(* CODESYS project CtaAppModBus_2.0.0.3.library
   Description: Modbus Library der CTA
   Version: 2.0.0.3
   Title: CtaAppModbus
   Author: SIS
   Company: CTA
   Placeholder: CtaAppModbus
   DocFormat: reStructuredText
   CompiledLibraryCompatibilityVersion: CODESYS V3.5 SP16 Patch 3
   LanguageModelAttribute: qualified-access-only
   DefaultNamespace: CtaAppModbus

Project tree, tasks and I/O mapping:
  libraries: Standard, 3.5.18.0 (System); CtaVisSymbols, 2.0.0.1 (CTA); CtaSysConfig, 2.0.0.0 (CTA); CtaAppTime, 2.0.0.0 (CTA); CtaAppBmk, 2.0.0.0 (CTA); VisuSymbols, 4.5.0.0 (System); VisuDialogs, * (System); ModbusFB, 4.5.0.0 (CODESYS); CtaVisUser, 1.0.0.0 (CTA); Util, 3.5.19.0 (System)
  10 Documenation/
    global variables VersionHistory
    global variables readMe
  00000000-0000-0000-0000-000000000000|D:\CoDeSys\LibrariesV3\trunk\Intern\CAA\CAA Template\3.4.0.0 draft\Placeholder.xml
  00000000-0000-0000-0000-000000000000|D:\CoDeSys\LibrariesV3\trunk\Intern\CAA\CAA Template\3.2.0.3 draft\Prefix.pdf
  00000000-0000-0000-0000-000000000000|D:\CoDeSys\LibrariesV3\trunk\Intern\CAA\CAA Template\3.5.2.0 draft\Placeholder.xml
  20 Structs/
    CLIENT/
      NETWORK/
        data type scTcpClientParameter
      SERIAL/
        data type scSerialPortParameter
        data type scSerialClientParameter
    SERVER/
      PARAMETER/
        SERIAL/
          data type scSerial
        data type scModBusServerParameter
        TCP/
          data type scTcp
  21 Interface/
    CLIENTMANAGER/
      BASE/
        interface ITF_MB_CLIENTMANAGER: AY_ITF_MBCLIENT_VIS, ITF_BASE_CLIENT, OperationTime, RELOAD_ARRAY
      RTU/
        interface ITF_MB_CLIENTMANAGER_RTU: P_fbbyDataBits, P_fbdwBaudrate, P_fbenDTRControl, P_fbenParity, P_fbenPort, P_fbenStopBits, P_fbenRTSControl, P_fbxRtuAscii
      TCP/
        interface ITF_MB_CLIENTMANAGER_TCP
    MBJOB/
      interface ITF_MBJOB: DESTROY, PARENT, pByte, SELF, BIG_SYBIL, byMbFunction, LOW_SYBIL, wMbAdress, wQuantity
    CLIENT/
      TCP/
        interface ITF_MB_CLIENT_TCP: WRITE_DELAY, IP_ADRESS, NODE_ID, P_fbstIpAdress, P_fbtReadDelay, P_fbtTimeOut, P_fbtWriteDelay, P_fbuiPort, P_fbusiNodeId, P_fbxEnable, PORT, READ_DELAY, TIMEOUT, ConnectTcp, Connected, ClientTcp
      RTU/
        interface ITF_MB_CLIENT_RTU: TIMEOUT, WRITE_DELAY, NODE_ID, P_fbtReadDelay, P_fbtWriteDelay, P_fbusiNodeId, P_fbxEnable, P_fbtTimeOut, READ_DELAY
      BASE/
        interface ITF_CLIENT: AY_ITF_MBJOB_VIS, COUNT, CREATE_JOB, RELOAD_ARRAY, DESTROY_JOB, SELF, ERROR_ID, ERROR, AllJobsDone, ADD_MODBUS_JOB, CALL_AFTER_LAST_JOB_DONE, CHECK_IF_JOB_EXIST, BASE_MBJOB, ExecuteTime, EXEPTION_CODE, GET_NEXT_JOB, GET_READY, IsCurrentCall, LOW_SYBIL, BIG_SYBIL, CONFIRM_ALL_JOBS_DONE, ENABLE, DESTROY_ALL_JOBS_ACTIVE, DESTROY_ALL_JOBS_REQUEST
    SERVER/
      interface ITF_SERVER_INFO_PARA: P_Serial_fbxRtuAscii, P_Serial_fbbyDataBits, NoSerialAccesSince, P_Serial_fbenDTRControl, P_Serial_fbenParity, P_Serial_fbenStopBits, P_Serial_fbenPort, P_Serial_fbtWatchDog, P_Serial_fbenRTSControl, P_Serial_fbxEnableWatchDog, P_Serial_fbusiNodeId, P_Serial_fbxEnable, P_Serial_fbdwBaudrate, TimeOutSerialWatchDog, RequestDataSerial, NoTcpAccesSince, P_Tcp_fbstInterface, P_Tcp_fbtWatchDog, P_Tcp_fbxEnable, P_Tcp_fbxEnableWatchDog, RequestDataTcp, TimeOutTcpWatchDog, P_Tcp_fbwPort, P_LoggingOp
      interface ITF_SERVER: metSetInputRegister, metSetHoldingRegister, metGetCoil, metGetHoldingRegister, metSetCoil, metSetDiscretInput
  30 Program Organization Units/
    FC/
      function fcStringIPtoByteArray [ST]
      function fcCheckIp [ST]
      function FcBytePointToBoolValue [ST]
      function FcBytePointToWordValue [ST]
      function fcSetInitialIPString [ST]
    CLIENT/
      BASE/
        function block FB_MB_CLIENT [ST]: ENABLE, ADD_MODBUS_JOB, COUNT, CREATE_JOB, DESTROY_JOB, ERROR, BIG_SYBIL, CALL_AFTER_LAST_JOB_DONE, CHECK_IF_JOB_EXIST, CONFIRM_ALL_JOBS_DONE, AllJobsDone, AY_ITF_MBJOB_VIS, BASE_MBJOB, ERROR_ID, ExecuteTime, EXEPTION_CODE, GET_NEXT_JOB, GET_READY, IsCurrentCall, LOW_SYBIL, RELOAD_ARRAY, SELF, DESTROY_ALL_JOBS_REQUEST, DESTROY_ALL_JOBS_ACTIVE, DESTROY_ALL_JOBS
      RTU/
        function block FB_MB_CLIENT_RTU [ST]: actConfig, ENABLE, NODE_ID, P_fbtReadDelay, P_fbtTimeOut, P_fbtWriteDelay, P_fbusiNodeId, P_fbxEnable, READ_DELAY, TIMEOUT, WRITE_DELAY
      TCP/
        function block FB_MB_CLIENT_TCP [ST]: actConfig, ENABLE, IP_ADRESS, P_fbtTimeOut, P_fbtWriteDelay, P_fbuiPort, P_fbusiNodeId, P_fbxEnable, WRITE_DELAY, PORT, NODE_ID, P_fbstIpAdress, READ_DELAY, P_fbtReadDelay, TIMEOUT, ConnectTcp, Connected, ClientTcp
        function block FB_MB_CLIENT_TCP_1 [ST]: actConfig, ENABLE, IP_ADRESS, P_fbtReadDelay, P_fbtTimeOut, P_fbtWriteDelay, P_fbuiPort, P_fbusiNodeId, P_fbxEnable, WRITE_DELAY, PORT, NODE_ID, P_fbstIpAdress, READ_DELAY, TIMEOUT
    SERVER/
      function block FB_SERVER [ST]: actConfig, actDataModel, actSerial, actTcp, metGetCoil, metGetHoldingRegister, metSetCoil, metSetDiscretInput, metSetHoldingRegister, metSetInputRegister, P_Serial_fbxEnableWatchDog, P_Serial_fbxRtuAscii, NoSerialAccesSince, P_Serial_fbbyDataBits, P_Serial_fbdwBaudrate, P_Serial_fbenDTRControl, P_Serial_fbenParity, P_Serial_fbenPort, P_Serial_fbenRTSControl, P_Serial_fbenStopBits, P_Serial_fbtWatchDog, P_Serial_fbusiNodeId, P_Serial_fbxEnable, RequestDataSerial, TimeOutSerialWatchDog, TimeOutTcpWatchDog, P_Tcp_fbwPort, P_Tcp_fbxEnable, P_Tcp_fbxEnableWatchDog, RequestDataTcp, NoTcpAccesSince, P_Tcp_fbstInterface, P_Tcp_fbtWatchDog, P_LoggingOp
      function block fbModBusServer [ST]: actConfig, actModBusServerSerial, actModBusServerTcp, actModBusServerUdp, metAddSerialControll, metAddTcpControll, metAddUdpControll, metGetCoil, metGetHoldingRegister, metSetCoil, metSetDiscretInput, metSetHoldingRegister, metSetInputRegister
      Serial/
        function block ServerSerial_Extended [ST]: RequestData, ProcessMaskWriteRegister, ProcessReadCoils, ProcessReadDiscreteInputs, ProcessReadHoldingRegisters, ProcessReadInputRegisters, ProcessReadWriteMultipleRegisters, ProcessWriteMultipleCoils, ProcessWriteMultipleRegisters, ProcessWriteSingleCoil, ProcessWriteSingleRegister
      Tcp/
        function block ServerTCP_Extended [ST]: RequestData, ProcessMaskWriteRegister, ProcessReadCoils, ProcessReadDiscreteInputs, ProcessReadHoldingRegisters, ProcessReadInputRegisters, ProcessReadWriteMultipleRegisters, ProcessWriteMultipleCoils, ProcessWriteMultipleRegisters, ProcessWriteSingleCoil, ProcessWriteSingleRegister
    MBJOB/
      function block FB_MBJOB [ST]: wMbAdress, BIG_SYBIL, wQuantity, SELF, byMbFunction, DESTROY, LOW_SYBIL, PARENT, pByte
    CLIENTMANAGER/
      RTU/
        function block FB_MB_CLIENTMANAGER_RTU [ST]: actCallFunctions, actDelays, actConfig, actExecuteFunction, actGetError, P_fbbyDataBits, P_fbdwBaudrate, P_fbenDTRControl, P_fbenParity, P_fbenRTSControl, P_fbenStopBits, P_fbxRtuAscii, P_fbenPort, actCheckBusy
      TCP/
        function block FB_MB_CLIENTMANAGER_TCP [ST]: actCallFunctions, actCheckBusy, actDelays, actExecuteFunction, actGetError
        function block FB_MB_CLIENTMANAGER_TCP_1 [ST]: actCallFunctions, actCheckBusy, actDelays, actExecuteFunction, actGetError
      BASE/
        function block FB_MB_CLIENTMANAGER [ST]: RELOAD_ARRAY, ADD_MODBUS_CLIENT, CHECK_IF_EXIST, AY_ITF_MBCLIENT_VIS, ITF_BASE_CLIENT, OperationTime, COUNT_ENABLED
  40 Visualizations/
    CLIENT/
      CLIENT/
        visualisation DIA_CLIENT
        JOBS/
          visualisation VIS_CLIENT_JOBS
          visualisation VIS_CLIENT_JOBS_QUERRY
          visualisation VIS_CLIENT_JOBS_TABLE
        MENÜ/
          visualisation VIS_CLIENT_MENÜ
        OVERWIEV/
          visualisation VIS_CLIENT_OVERWIEV
          visualisation VIS_CLIENT_OVERWIEV_QUERY
        PARAMETER/
          visualisation VIS_CLIENT_PARAMETER
      RTU/
        PARAMETER/
          visualisation VIS_CLIENT_PARAMETER_RTU_QUERY
          visualisation VIS_CLIENT_PARAMETER_RTU
          visualisation VIS_CLIENT_PARAMETER_RTU_TEMP
      TCP/
        PARAMETER/
          visualisation VIS_CLIENT_PARAMETER_TCP
          visualisation VIS_CLIENT_PARAMETER_TCP_TEMP
          visualisation VIS_CLIENT_PARAMETER_TCP_QUERY
    TEXTLIST/
      text list TEXT_DTR_CONTROL
      text list TEXT_PARITY
      text list TEXT_RTS_CONTROL
      text list TEXT_STOPBITS
      text list TXT_COMPORT
    CLIENTMANAGER/
      visualisation DIA_CLIENT_MANAGER
      LINE/
        visualisation VIS_CLIENT_LINE
        visualisation VIS_CLIENT_LINE_QUERRY
      MENÜ/
        visualisation VIS_CLIENTMANAGER_MENÜ
      OVERWIEV/
        visualisation VIS_CLIENT_MANAGER_OVERWIEV
        visualisation VIS_CLIENT_MANAGER_OVERWIEV_QUERRY
        visualisation VIS_CLIENT_MANAGER_TABLE
      PARAMETER/
        visualisation VIS_CLIENT_MANAGER_PARAMETER
      RTU/
        PARAMETER/
          visualisation VIS_CLIENT_MANAGER_PARAMETER_RTU
          visualisation VIS_CLIENT_MANAGER_PARAMETER_RTU_QUERY
          visualisation VIS_CLIENT_MANAGER_PARAMETER_RTU_TEMP
      TCP/
        PARAMETER/
          visualisation VIS_CLIENT_MANAGER_PARAMETER_TCP
          visualisation VIS_CLIENT_MANAGER_PARAMETER_TCP_QUERY
    HELPER/
      visualisation VIS_IP_PARAMETER
      visualisation DIA_IP_INPUT
      visualisation VIS_IP_PARAMETER_QUERRY
      visualisation VIS_IP_PARAMETER_BASE
    MBJOB/
      visualisation VIS_JOB
      visualisation VIS_JOB_QUERRY
    SERVER/
      visualisation DIA_SERVER
      SERIAL/
        visualisation VIS_SERVER_SERIAL_STATE
        visualisation VIS_SERVER_SERIAL_STATE_INFO
        PARAMETER/
          visualisation DIA_SERVER_SERIAL_PARAMETER
          visualisation VIS_SERVER_SERIAL_PARAMETER
      TCP/
        visualisation VIS_SERVER_TCP_STATE
        visualisation VIS_SERVER_TCP_STATE_INFO
        PARAMETER/
          visualisation DIA_SERVER_TCP_PARAMETER
          visualisation VIS_SERVER_TCP_PARAMETER
  text list GlobalTextList
  60 Textlisten/
    SERIAL/
      text list txtHandshake
      text list txtParity
      text list txtPhysikalLayer
      text list txtStopBits
    text list txtLoggingOp
*)

// 20 Structs/CLIENT/SERIAL/scSerialPortParameter
TYPE scSerialPortParameter :
    STRUCT 
		fbenPort							:	CtaSysConfig.fbINT;			// PORT NONE , COM1, COM2 ...
		fbdwBaudrate						:	CtaSysConfig.fbDWORD;		// Baudrate 
		fbbyDataBits						:	CtaSysConfig.fbBYTE;		// Data Bits
		fbenParity							:	CtaSysConfig.fbBYTE;		// Parity
		fbenStopBits						:	CtaSysConfig.fbBYTE;		// Stopbits
		fbenDTRControl						:	CtaSysConfig.fbBYTE;		// DTR Control
		fbenRTSControl						:	CtaSysConfig.fbBYTE;		// RTS Control
		fbxRtuAscii							:	CtaSysConfig.fbBOOL;		// RTU = FALSE , ASCII = TRUE
    END_STRUCT
END_TYPE

// 20 Structs/CLIENT/SERIAL/scSerialClientParameter
TYPE scSerialClientParameter :
    STRUCT
        fbxEnable					:	CtaSysConfig.fbBOOL;       // Serial Server Enable        
        fbusiNodeId					:	CtaSysConfig.fbUSINT;      // Serial Server Id        
        fbtTimeOut					:	CtaSysConfig.fbTIME;       // Timeout Time
		fbtReadDelay				:	CtaSysConfig.fbTIME; 	   // Read Delay
		fbtWriteDelay				:	CtaSysConfig.fbTIME;	   // Write Delay
    END_STRUCT
END_TYPE

// 20 Structs/SERVER/PARAMETER/SERIAL/scSerial
TYPE scSerial :
    STRUCT
        fbxEnable           				:   CtaSysConfig.fbBOOL;        // Serial Server Enable
        fbxEnableWatchDog   				:   CtaSysConfig.fbBOOL;        // WatchDog Enable
        fbtWatchDog         				:   CtaSysConfig.fbTIME;        // WatchDog Time		
		fbenPort							:	CtaSysConfig.fbINT;			// PORT NONE , COM1, COM2 ...
		fbusiNodeId							:	CtaSysConfig.fbUSINT;      	// Serial Server Id  
		fbdwBaudrate						:	CtaSysConfig.fbDWORD;		// Baudrate 
		fbbyDataBits						:	CtaSysConfig.fbBYTE;		// Data Bits
		fbenParity							:	CtaSysConfig.fbBYTE;		// Parity
		fbenStopBits						:	CtaSysConfig.fbBYTE;		// Stopbits
		fbenDTRControl						:	CtaSysConfig.fbBYTE;		// DTR Control
		fbenRTSControl						:	CtaSysConfig.fbBYTE;		// RTS Control
		fbxRtuAscii							:	CtaSysConfig.fbBOOL;		// RTU = FALSE , ASCII = TRUE
    END_STRUCT
END_TYPE

// 20 Structs/SERVER/PARAMETER/TCP/scTcp
TYPE scTcp :
    STRUCT
        fbxEnable           :   CtaSysConfig.fbBOOL;           // Tcp Server Enable    
        fbwPort             :   CtaSysConfig.fbWORD;           // Tcp Server Port
        fbxEnableWatchDog   :   CtaSysConfig.fbBOOL;           // WatchDog Enable
        fbtWatchDog         :   CtaSysConfig.fbTIME;           // WatchDog Time
		fbstInterface		:	CtaSysConfig.fbSTRING40;	   // Interface Name
    END_STRUCT
END_TYPE

// 20 Structs/CLIENT/NETWORK/scTcpClientParameter
TYPE scTcpClientParameter :
    STRUCT
        fbxEnable					:	CtaSysConfig.fbBOOL;        // Serial Server Enable       
        fbusiNodeId					:	CtaSysConfig.fbUSINT;     	// Serial Server Id  
        fbtTimeOut					:	CtaSysConfig.fbTIME;        // Timeout Time
        fbtReadDelay				:	CtaSysConfig.fbTIME;      	// Read Delay        
        fbtWriteDelay				:	CtaSysConfig.fbTIME;     	// Write Delay 	
		fbuiPort					:	CtaSysConfig.fbUINT;      	// Port Nr  
		fbstIpAdress				:	CtaSysConfig.fbSTRING40;    // IP Adresse   
    END_STRUCT
END_TYPE

// 20 Structs/SERVER/PARAMETER/scModBusServerParameter
TYPE scModBusServerParameter :
    STRUCT
        scSerial    :   scSerial;
        scTcp       :   scTcp;
		loggingOp	:	CtaSysConfig.fbDWORD;
    END_STRUCT
END_TYPE

// 10 Documenation/VersionHistory
(* 

.. image:: ../../Images/CTA_Logo.jpg
   :align: right
   :width: 15% 

**Vorlage**   


============ =========== =========== ============================================
**Date**     **Version** **Author**  **Change**
------------ ----------- ----------- --------------------------------------------
04.03.2021   0.0.0.0     SIS         Vorlage erstellt

============ =========== =========== ============================================


*)
VAR_GLOBAL
    stInfo : STRING:= '0.0.0.0, Vorlage, CTA';
END_VAR

// 10 Documenation/readMe
(*

**ReadMe**
 
|	**Empfehlung**
|
|	Dokumentrieren Sie die Library für eine nachhaltige Entwicklung
|     
| *Beispiel* 
|
| Dies ist die Vorlage Library der CTA. Erstellen Sie ihre Library anhand dieser Vorlage.
*)

VAR_GLOBAL
    xReadMeDone              :   BOOL;
END_VAR

// 21 Interface/SERVER/ITF_SERVER_INFO_PARA
INTERFACE ITF_SERVER_INFO_PARA EXTENDS ITF_SERVER

PROPERTY P_Serial_fbxRtuAscii : CtaSysConfig.ITF_BOOL
GET
END_GET
END_PROPERTY

PROPERTY P_Serial_fbbyDataBits : CtaSysConfig.ITF_BYTE
GET
END_GET
END_PROPERTY

PROPERTY NoSerialAccesSince : TIME
GET
END_GET
END_PROPERTY

PROPERTY P_Serial_fbenDTRControl : CtaSysConfig.ITF_BYTE
GET
END_GET
END_PROPERTY

PROPERTY P_Serial_fbenParity : CtaSysConfig.ITF_BYTE
GET
END_GET
END_PROPERTY

PROPERTY P_Serial_fbenStopBits : CtaSysConfig.ITF_BYTE
GET
END_GET
END_PROPERTY

PROPERTY P_Serial_fbenPort : CtaSysConfig.ITF_INT
GET
END_GET
END_PROPERTY

PROPERTY P_Serial_fbtWatchDog : CtaSysConfig.ITF_TIME
GET
END_GET
END_PROPERTY

PROPERTY P_Serial_fbenRTSControl : CtaSysConfig.ITF_BYTE
GET
END_GET
END_PROPERTY

PROPERTY P_Serial_fbxEnableWatchDog : CtaSysConfig.ITF_BOOL
GET
END_GET
END_PROPERTY

PROPERTY P_Serial_fbusiNodeId : CtaSysConfig.ITF_USINT
GET
END_GET
END_PROPERTY

PROPERTY P_Serial_fbxEnable : CtaSysConfig.ITF_BOOL
GET
END_GET
END_PROPERTY

PROPERTY P_Serial_fbdwBaudrate : CtaSysConfig.ITF_DWORD
GET
END_GET
END_PROPERTY

PROPERTY TimeOutSerialWatchDog : BOOL
GET
END_GET
END_PROPERTY

PROPERTY RequestDataSerial : String
GET
END_GET
END_PROPERTY

PROPERTY NoTcpAccesSince : TIME
GET
END_GET
END_PROPERTY

PROPERTY P_Tcp_fbstInterface : CtaSysConfig.ITF_STRING40
GET
END_GET
END_PROPERTY

PROPERTY P_Tcp_fbtWatchDog : CtaSysConfig.ITF_TIME
GET
END_GET
END_PROPERTY

PROPERTY P_Tcp_fbxEnable : CtaSysConfig.ITF_BOOL
GET
END_GET
END_PROPERTY

PROPERTY P_Tcp_fbxEnableWatchDog : CtaSysConfig.ITF_BOOL
GET
END_GET
END_PROPERTY

PROPERTY RequestDataTcp : STRING
GET
END_GET
END_PROPERTY

PROPERTY TimeOutTcpWatchDog : BOOL
GET
END_GET
END_PROPERTY

PROPERTY P_Tcp_fbwPort : CtaSysConfig.ITF_WORD
GET
END_GET
END_PROPERTY

PROPERTY P_LoggingOp : CtaSysConfig.ITF_DWORD
GET
END_GET
END_PROPERTY

END_INTERFACE

// 21 Interface/SERVER/ITF_SERVER
INTERFACE ITF_SERVER EXTENDS __SYSTEM.IQueryInterface

METHOD metSetInputRegister : BOOL
VAR_INPUT
    wAdr          : WORD;
    wValue        : WORD;
END_VAR
END_METHOD

METHOD metSetHoldingRegister : BOOL
VAR_INPUT
    wAdr          : WORD;
    wValue        : WORD;
END_VAR
END_METHOD

METHOD metGetCoil : BOOL
VAR_INPUT
    wAdr          : WORD;
END_VAR
END_METHOD

METHOD metGetHoldingRegister : WORD
VAR_INPUT
    wAdr          : WORD;
END_VAR
END_METHOD

METHOD metSetCoil : BOOL
VAR_INPUT
    wAdr          : WORD;
    xValue        : BOOL;
END_VAR
END_METHOD

METHOD metSetDiscretInput : BOOL
VAR_INPUT
    wAdr          : WORD;
    xValue        : BOOL;
END_VAR
END_METHOD

END_INTERFACE

// 21 Interface/CLIENTMANAGER/BASE/ITF_MB_CLIENTMANAGER
INTERFACE ITF_MB_CLIENTMANAGER EXTENDS CtaAppBmk.ITF_BMK

PROPERTY AY_ITF_MBCLIENT_VIS : ARRAY[0..9] OF ITF_CLIENT
GET
END_GET
END_PROPERTY

PROPERTY ITF_BASE_CLIENT : ITF_CLIENT
GET
END_GET
END_PROPERTY

PROPERTY OperationTime : LTIME
GET
END_GET
END_PROPERTY

METHOD RELOAD_ARRAY
VAR_INPUT
	xInit				:	BOOL;
	xLoadNext10			:	BOOL;
	xLoadLast10			:	BOOL;
END_VAR
END_METHOD

END_INTERFACE

// 21 Interface/CLIENT/BASE/ITF_CLIENT
INTERFACE ITF_CLIENT  EXTENDS CtaAppBmk.ITF_BMK

PROPERTY AY_ITF_MBJOB_VIS : ARRAY[0..9] OF ITF_MBJOB
GET
END_GET
END_PROPERTY

PROPERTY COUNT : UINT
GET
END_GET
END_PROPERTY

METHOD CREATE_JOB : BOOL
VAR_INPUT
	_byMbFunction	:	BYTE;
	_wMbAdress		:	WORD;
	_pData			:	POINTER TO BYTE;
	_wQuantity		:	WORD;		
END_VAR
END_METHOD

METHOD RELOAD_ARRAY
VAR_INPUT
	xInit				:	BOOL;
	xLoadNext10			:	BOOL;
	xLoadLast10			:	BOOL;
END_VAR
END_METHOD

METHOD DESTROY_JOB : BOOL
VAR_INPUT
	_byMbFunction	:	BYTE;
	_wMbAdress		:	WORD;
	_pData			:	POINTER TO BYTE;
	_wQuantity		:	WORD;		
END_VAR
END_METHOD

PROPERTY SELF : ITF_CLIENT
GET
END_GET
END_PROPERTY

PROPERTY ERROR_ID : ModbusFB.Error
GET
END_GET
SET
END_SET
END_PROPERTY

PROPERTY ERROR : BOOL
GET
END_GET
SET
END_SET
END_PROPERTY

PROPERTY AllJobsDone : BOOL
GET
END_GET
END_PROPERTY

METHOD ADD_MODBUS_JOB
VAR_INPUT
	ITF_MBJOB_IN	:	ITF_MBJOB;
END_VAR
END_METHOD

METHOD CALL_AFTER_LAST_JOB_DONE
VAR_INPUT
END_VAR
END_METHOD

METHOD CHECK_IF_JOB_EXIST : BOOL
VAR_INPUT
	_byMbFunction	:	BYTE;
	_wMbAdress		:	WORD;
	_pByte			:	POINTER TO BYTE;
	_wQuantity		:	WORD;	
END_VAR
END_METHOD

PROPERTY BASE_MBJOB : ITF_MBJOB
GET
END_GET
END_PROPERTY

PROPERTY ExecuteTime : LTIME
GET
END_GET
END_PROPERTY

PROPERTY EXEPTION_CODE : ModbusFB.ExceptionCodes
GET
END_GET
SET
END_SET
END_PROPERTY

METHOD GET_NEXT_JOB : BOOL
VAR_OUTPUT
	_byMbFunction	:	BYTE;
	_wMbAdress		:	WORD;
	_pByte			:	POINTER TO BYTE;
	_wQuantity		:	WORD;	
END_VAR
END_METHOD

METHOD GET_READY : BOOL
VAR_INPUT
END_VAR
END_METHOD

PROPERTY IsCurrentCall : BOOL
GET
END_GET
END_PROPERTY

PROPERTY LOW_SYBIL : ITF_CLIENT
SET
END_SET
GET
END_GET
END_PROPERTY

PROPERTY BIG_SYBIL : ITF_CLIENT
GET
END_GET
SET
END_SET
END_PROPERTY

PROPERTY CONFIRM_ALL_JOBS_DONE : BOOL
GET
END_GET
END_PROPERTY

PROPERTY ENABLE : BOOL
GET
END_GET
END_PROPERTY

PROPERTY DESTROY_ALL_JOBS_ACTIVE : BOOL
GET
END_GET
END_PROPERTY

METHOD DESTROY_ALL_JOBS_REQUEST
VAR_INPUT
END_VAR
END_METHOD

END_INTERFACE

// 21 Interface/MBJOB/ITF_MBJOB
INTERFACE ITF_MBJOB EXTENDS __System.IQUERYINTERFACE

METHOD DESTROY
END_METHOD

PROPERTY PARENT : ITF_CLIENT
SET
END_SET
END_PROPERTY

PROPERTY pByte : POINTER TO BYTE
GET
END_GET
SET
END_SET
END_PROPERTY

PROPERTY SELF : ITF_MBJOB
GET
END_GET
END_PROPERTY

PROPERTY BIG_SYBIL : ITF_MBJOB
GET
END_GET
SET
END_SET
END_PROPERTY

PROPERTY byMbFunction : BYTE
GET
END_GET
SET
END_SET
END_PROPERTY

PROPERTY LOW_SYBIL : ITF_MBJOB
GET
END_GET
SET
END_SET
END_PROPERTY

PROPERTY wMbAdress : WORD
GET
END_GET
SET
END_SET
END_PROPERTY

PROPERTY wQuantity : WORD
GET
END_GET
SET
END_SET
END_PROPERTY

END_INTERFACE

// 21 Interface/CLIENTMANAGER/RTU/ITF_MB_CLIENTMANAGER_RTU
INTERFACE ITF_MB_CLIENTMANAGER_RTU EXTENDS ITF_MB_CLIENTMANAGER

PROPERTY P_fbbyDataBits : CtaSysConfig.ITF_DATATYPE
GET
END_GET
END_PROPERTY

PROPERTY P_fbdwBaudrate : CtaSysConfig.ITF_DATATYPE
GET
END_GET
END_PROPERTY

PROPERTY P_fbenDTRControl : CtaSysConfig.ITF_BYTE
GET
END_GET
END_PROPERTY

PROPERTY P_fbenParity : CtaSysConfig.ITF_BYTE
GET
END_GET
END_PROPERTY

PROPERTY P_fbenPort : CtaSysConfig.ITF_INT
GET
END_GET
END_PROPERTY

PROPERTY P_fbenStopBits : CtaSysConfig.ITF_BYTE
GET
END_GET
END_PROPERTY

PROPERTY P_fbenRTSControl : CtaSysConfig.ITF_BYTE
GET
END_GET
END_PROPERTY

PROPERTY P_fbxRtuAscii : CtaSysConfig.ITF_DATATYPE
GET
END_GET
END_PROPERTY

END_INTERFACE

// 21 Interface/CLIENT/TCP/ITF_MB_CLIENT_TCP
INTERFACE ITF_MB_CLIENT_TCP  EXTENDS ITF_CLIENT

PROPERTY WRITE_DELAY : TIME
GET
END_GET
END_PROPERTY

PROPERTY IP_ADRESS : STRING(15)
GET
END_GET
END_PROPERTY

PROPERTY NODE_ID : USINT
GET
END_GET
END_PROPERTY

PROPERTY P_fbstIpAdress : CtaSysConfig.ITF_DATATYPE
GET
END_GET
END_PROPERTY

PROPERTY P_fbtReadDelay : CtaSysConfig.ITF_DATATYPE
GET
END_GET
END_PROPERTY

PROPERTY P_fbtTimeOut : CtaSysConfig.ITF_DATATYPE
GET
END_GET
END_PROPERTY

PROPERTY P_fbtWriteDelay : CtaSysConfig.ITF_DATATYPE
GET
END_GET
END_PROPERTY

PROPERTY P_fbuiPort : CtaSysConfig.ITF_DATATYPE
GET
END_GET
END_PROPERTY

PROPERTY P_fbusiNodeId : CtaSysConfig.ITF_DATATYPE
GET
END_GET
END_PROPERTY

PROPERTY P_fbxEnable : CtaSysConfig.ITF_DATATYPE
GET
END_GET
END_PROPERTY

PROPERTY PORT : UINT
GET
END_GET
END_PROPERTY

PROPERTY READ_DELAY : TIME
GET
END_GET
END_PROPERTY

PROPERTY TIMEOUT : TIME
GET
END_GET
END_PROPERTY

METHOD ConnectTcp : BOOL
VAR_INPUT
END_VAR
END_METHOD

PROPERTY Connected : BOOL
GET
END_GET
END_PROPERTY

PROPERTY  ClientTcp : REFERENCE TO ModbusFB.Client
GET
END_GET
END_PROPERTY

END_INTERFACE

// 30 Program Organization Units/FC/fcStringIPtoByteArray
FUNCTION fcStringIPtoByteArray : ARRAY[0..3] OF BYTE
VAR_INPUT
	stIP	:	STRING;
END_VAR
VAR
    temp_string 	: STRING;
    dot_pos 		: INT;
    i 				: INT;
    part 			: STRING[4];
    value 			: WORD;
END_VAR

temp_string := stIP;
REPEAT
    dot_pos := FIND(temp_string,'.');
    IF dot_pos > 0 THEN
        part := LEFT(temp_string, dot_pos - 1);
        temp_string := RIGHT(temp_string, LEN(temp_string) - dot_pos);
    ELSE
        part := temp_string;
    END_IF

    // Umwandeln in BYTE
    value := STRING_TO_WORD(part);
    IF (value >= 0) AND (value <= 255) THEN
        fcStringIPtoByteArray[i] := WORD_TO_BYTE(value);
    ELSE
        RETURN;
    END_IF

    i := i + 1;
UNTIL (dot_pos = 0) OR (i > 3)
END_REPEAT

// Setze auf 0 wenn nicht 4 Segmente gefunden wurden
IF i <> 4 THEN
	fcStringIPtoByteArray[0] := 0;
	fcStringIPtoByteArray[1] := 0;
	fcStringIPtoByteArray[2] := 0;
	fcStringIPtoByteArray[3] := 0;
END_IF

END_FUNCTION

// 30 Program Organization Units/FC/fcCheckIp
FUNCTION fcCheckIp : BOOL
VAR_INPUT
    stIp           : STRING[20];
END_VAR
VAR
    iFor           : INT;
    iCountPacket   : INT;
    iCountPoint    : INT;
    iCountZiffer   : INT;
    xFail          : BOOL;
END_VAR

FOR iFor := LEN(stIp) TO 0 BY -1 DO
    // Check Termination
    IF iFor = LEN(stIp) THEN
        IF stIp[iFor] <> 0 THEN 
            xFail := TRUE; // No Termination
            EXIT;       
        END_IF;
	ELSE
        // Check if Ziffer
        IF stIp[iFor] >= 48 AND stIp[iFor] <= 57 THEN    
            IF iCountZiffer < 3 THEN
                IF iCountZiffer = 0 THEN
                    IF iFor >= 2 THEN
                        IF stIp[iFor - 2] >= 50 THEN
                            // Check if Ziffer <= 5
                            IF stIp[iFor] <= 53 THEN     
                                iCountZiffer := iCountZiffer + 1;
                            ELSE
                                xFail := TRUE;  // Max is 255
                                EXIT;
                            END_IF;   
                        ELSE
                            iCountZiffer := iCountZiffer + 1;                   
						END_IF;                        
                    ELSE
                        iCountZiffer := iCountZiffer + 1;
					END_IF
                ELSIF iCountZiffer = 1 THEN
                    IF iFor <> 0 THEN
                        IF stIp[iFor - 1] = 46 THEN
                            iCountZiffer := iCountZiffer + 1;
                        // Check if next Ziffer is 2    
                        ELSIF stIp[iFor - 1] >= 50 THEN  
                            // Check if Ziffer <= 5
                            IF stIp[iFor] <= 53 THEN     
                                iCountZiffer := iCountZiffer + 1;
                            ELSE
                                xFail := TRUE;  // Max is 255
                                EXIT;
                            END_IF;    
                        END_IF;
                    ELSE
                        iCountZiffer := iCountZiffer + 1;        
					END_IF;                       
                ELSIF iCountZiffer = 2 THEN
                    IF stIp[iFor] <= 50 THEN
                        iCountZiffer := iCountZiffer + 1;
                    ELSE
                        xFail := TRUE;
                        EXIT;
					END_IF
                END_IF;    
            ELSIF iCountZiffer = 3 THEN
                xFail := TRUE; // More Then 3 Ziffers not allowed!
                EXIT;
            END_IF;
        // Check if Point
        ELSIF stIp[iFor] = 46 THEN
            IF iCountZiffer > 0 THEN
                iCountPacket := iCountPacket + 1;
                iCountPoint  := iCountPoint + 1;
                iCountZiffer := 0;
            ELSE
                xFail := TRUE; // Empty Packet not allowed!
                EXIT;
            END_IF;   
        END_IF;
    END_IF;
END_FOR;

IF xFail THEN
    fcCheckIp := FALSE;
ELSIF iCountPoint = 3 AND iCountPacket = 3 AND iCountZiffer > 0 THEN    
    fcCheckIp := TRUE;
END_IF;

END_FUNCTION

// 30 Program Organization Units/CLIENTMANAGER/TCP/FB_MB_CLIENTMANAGER_TCP
{attribute 'no_assign'}
FUNCTION_BLOCK FB_MB_CLIENTMANAGER_TCP EXTENDS FB_MB_CLIENTMANAGER IMPLEMENTS ITF_MB_CLIENTMANAGER_TCP
VAR_OUTPUT
END_VAR
VAR
	_TEMP_MBU_CLIENT_TCP				:	ITF_MB_CLIENT_TCP;
	
	fbReadCoilsFc01						:	ModbusFB.ClientRequestReadCoils;
	fbReadDiscreteInputsFc02			:	ModbusFB.ClientRequestReadDiscreteInputs;
	fbReadHoldingRegistersFc03			:	ModbusFB.ClientRequestReadHoldingRegisters;
	fbReadInputRegistersFc04			:	ModbusFB.ClientRequestReadInputRegisters;
	fbWriteSingleCoilFc05				:	ModbusFB.ClientRequestWriteSingleCoil;
	fbWriteSingleRegisterFc06			:	ModbusFB.ClientRequestWriteSingleRegister;
	fbWriteMultipleCoilsFc15			:	ModbusFB.ClientRequestWriteMultipleCoils;
	fbWriteMultipleRegistersFc16		:	ModbusFB.ClientRequestWriteMultipleRegisters;
	
END_VAR

SUPER^();
(* Check if one is allready Working *)
IF NOT xIsWorking THEN
	(* Get Client Ready *)
	IF __QUERYINTERFACE(_TEMP_MBU_CLIENT,_TEMP_MBU_CLIENT) THEN
		xIsWorking 		:= TRUE;	
		xErrorHappen	:= FALSE;
		eErrorID		:= ModbusFB.Error.OK;
		eExeptionCode	:= ModbusFB.ExceptionCodes.RESPONSE_SUCCESS;		
	(* Get Base Client Ready *)
	ELSIF __QUERYINTERFACE(_BASE_MBU_CLIENT,_TEMP_MBU_CLIENT) THEN
		xIsWorking 		:= TRUE;
		xErrorHappen	:= FALSE;
		eErrorID		:= ModbusFB.Error.OK;
		eExeptionCode	:= ModbusFB.ExceptionCodes.RESPONSE_SUCCESS;
		ltTime 			:= fbTimeStop.Stop();
		fbTimeStop.Start();
	END_IF;
END_IF;
(* Check if is running *)
IF xIsWorking THEN
	IF __QUERYINTERFACE(_TEMP_MBU_CLIENT,_TEMP_MBU_CLIENT) THEN	
		(* Wait until no Execute *)		
		IF 	NOT	fbReadCoilsFc01.xExecute				AND
			NOT	fbReadDiscreteInputsFc02.xExecute	    AND
			NOT	fbReadHoldingRegistersFc03.xExecute     AND
			NOT	fbReadInputRegistersFc04.xExecute	    AND
			NOT	fbWriteSingleCoilFc05.xExecute		    AND
			NOT	fbWriteSingleRegisterFc06.xExecute	    AND
			NOT	fbWriteMultipleCoilsFc15.xExecute	    AND
			NOT	fbWriteMultipleRegistersFc16.xExecute	THEN
			(* Get Type of Port *) 
			IF __QUERYINTERFACE(_TEMP_MBU_CLIENT,_TEMP_MBU_CLIENT_TCP) THEN
				(* Check if Enabled *)
				IF _TEMP_MBU_CLIENT_TCP.ENABLE AND _TEMP_MBU_CLIENT_TCP.COUNT > 0 THEN
					IF NOT _TEMP_MBU_CLIENT_TCP.IsCurrentCall THEN
						_TEMP_MBU_CLIENT_TCP.GET_READY();
						tTimeOut		:= _TEMP_MBU_CLIENT_TCP.TIMEOUT;
						tReadDelay		:= _TEMP_MBU_CLIENT_TCP.READ_DELAY;
						tWriteDelay	 	:= _TEMP_MBU_CLIENT_TCP.WRITE_DELAY;
					END_IF;
					(* Connect *)
					IF NOT _TEMP_MBU_CLIENT_TCP.Connected THEN
						xAbort 			:= _TEMP_MBU_CLIENT_TCP.ConnectTcp();
						usiNodeId 		:= _TEMP_MBU_CLIENT_TCP.NODE_ID;
					END_IF;
				ELSE
					xAbort		:= TRUE;
				END_IF;
			ELSE
				xAbort := TRUE;
			END_IF;
			(* Check if Connected *)
			IF _TEMP_MBU_CLIENT_TCP.Connected AND NOT xAbort THEN
				(* Get Job *)
				IF NOT xTrig THEN
					xTrig := _TEMP_MBU_CLIENT.GET_NEXT_JOB(_byMbFunction => _byMbFunction,_wMbAdress => _wMbAdress,_pByte => _pByte,_wQuantity => _wQuantity);
				END_IF;
				
				(* Delay Function *)
				actDelays();
				
				(* Execute Function *)
				actExecuteFunction();
				
				(* Resett Timer *)
				IF tonDelay.Q THEN
					tonDelay(IN := FALSE);
					xTrig := FALSE;
				END_IF;
			END_IF;
		ELSE
			(* Check Busy *)
			actCheckBusy();					
		END_IF;
		(* Get Errors *)
		actGetError();
		(* Check if All Job as Done *)
		IF _TEMP_MBU_CLIENT.AllJobsDone OR xAbort THEN
			(* Wait until no Execute *)		
			IF 	NOT xTrig									AND
				NOT	fbReadCoilsFc01.xExecute				AND
				NOT	fbReadDiscreteInputsFc02.xExecute	    AND
				NOT	fbReadHoldingRegistersFc03.xExecute     AND
				NOT	fbReadInputRegistersFc04.xExecute	    AND
				NOT	fbWriteSingleCoilFc05.xExecute		    AND
				NOT	fbWriteSingleRegisterFc06.xExecute	    AND
				NOT	fbWriteMultipleCoilsFc15.xExecute	    AND
				NOT	fbWriteMultipleRegistersFc16.xExecute	THEN
				_TEMP_MBU_CLIENT.CALL_AFTER_LAST_JOB_DONE();
				(* Set Error if Job > 0 *)
				IF _TEMP_MBU_CLIENT.COUNT > 0 THEN
					_TEMP_MBU_CLIENT.ERROR			:= xErrorHappen;
					_TEMP_MBU_CLIENT.ERROR_ID		:= eErrorID;
					_TEMP_MBU_CLIENT.EXEPTION_CODE	:= eExeptionCode;
				END_IF;
				_TEMP_MBU_CLIENT 					:= _TEMP_MBU_CLIENT.LOW_SYBIL;
				_byMbFunction 					:= 0;
				_wMbAdress	  					:= 0;
				_pByte		  					:= 0;
				_wQuantity						:= 0;
				xIsWorking						:= FALSE;
				xAbort							:= FALSE;
			END_IF;
		END_IF;
	END_IF;
END_IF;

(* Call Functions *)
actCallFunctions();

ACTION actCallFunctions:
(* Call *)
IF __QUERYINTERFACE(_TEMP_MBU_CLIENT_TCP,_TEMP_MBU_CLIENT_TCP) THEN
	fbReadCoilsFc01(				rClient := _TEMP_MBU_CLIENT_TCP.ClientTcp);		
	fbReadDiscreteInputsFc02(		rClient := _TEMP_MBU_CLIENT_TCP.ClientTcp);  
	fbReadHoldingRegistersFc03(		rClient := _TEMP_MBU_CLIENT_TCP.ClientTcp);
	fbReadInputRegistersFc04(		rClient := _TEMP_MBU_CLIENT_TCP.ClientTcp);	  
	fbWriteSingleCoilFc05(			rClient := _TEMP_MBU_CLIENT_TCP.ClientTcp);	  
	fbWriteSingleRegisterFc06(		rClient := _TEMP_MBU_CLIENT_TCP.ClientTcp);  
	fbWriteMultipleCoilsFc15(		rClient := _TEMP_MBU_CLIENT_TCP.ClientTcp);  
	fbWriteMultipleRegistersFc16(	rClient := _TEMP_MBU_CLIENT_TCP.ClientTcp);
END_IF;
END_ACTION

ACTION actCheckBusy:
(* Reset after Busy *)
fbReadCoilsFc01.xExecute				:= fbReadCoilsFc01.xBusy				;
fbReadDiscreteInputsFc02.xExecute	    := fbReadDiscreteInputsFc02.xBusy		;
fbReadHoldingRegistersFc03.xExecute     := fbReadHoldingRegistersFc03.xBusy		;
fbReadInputRegistersFc04.xExecute	    := fbReadInputRegistersFc04.xBusy		;
fbWriteSingleCoilFc05.xExecute		    := fbWriteSingleCoilFc05.xBusy			;
fbWriteSingleRegisterFc06.xExecute	    := fbWriteSingleRegisterFc06.xBusy		;
fbWriteMultipleCoilsFc15.xExecute	    := fbWriteMultipleCoilsFc15.xBusy		;
fbWriteMultipleRegistersFc16.xExecute   := fbWriteMultipleRegistersFc16.xBusy	;
END_ACTION

ACTION actDelays:
(* Delay Read *)
IF _byMbFunction <= 04 THEN
	tonDelay(IN := xTrig,PT := tReadDelay);
(* Delay Write Single *)
ELSIF _byMbFunction >= 5 AND _byMbFunction <= 6 THEN
	tonDelay(IN := xTrig,PT := tWriteDelay); 
(* Delay Write Multiple *)
ELSIF _byMbFunction >= 15 AND _byMbFunction <= 16 THEN
	tonDelay(IN := xTrig,PT := tWriteDelay); 
ELSE 
	tonDelay(IN := xTrig,PT := T#0MS);
END_IF;
END_ACTION

ACTION actExecuteFunction:
(* Read Coils *)
IF _byMbFunction = 01 THEN
	fbReadCoilsFc01.udiReplyTimeout					:= TO_UDINT(tTimeOut) * 1000; 
	fbReadCoilsFc01.udiTimeOut						:= TO_UDINT(tTimeOut) * 1000 * 2;
	fbReadCoilsFc01.uiUnitId						:= usiNodeId;
	fbReadCoilsFc01.uiStartItem 					:= TO_UINT(_wMbAdress);
	fbReadCoilsFc01.pData 							:= _pByte;
	fbReadCoilsFc01.uiQuantity						:= TO_UINT(_wQuantity);
	fbReadCoilsFc01.xExecute						:= tonDelay.Q;
(* Read Discret Inputs *)                       	
ELSIF _byMbFunction = 02 THEN                   	
	fbReadDiscreteInputsFc02.udiReplyTimeout		:= TO_UDINT(tTimeOut) * 1000; 
	fbReadDiscreteInputsFc02.udiTimeOut				:= TO_UDINT(tTimeOut) * 1000 * 2;
	fbReadDiscreteInputsFc02.uiUnitId				:= usiNodeId;
	fbReadDiscreteInputsFc02.uiStartItem			:= TO_UINT(_wMbAdress);
	fbReadDiscreteInputsFc02.pData 					:= _pByte;
	fbReadDiscreteInputsFc02.uiQuantity				:= TO_UINT(_wQuantity);
	fbReadDiscreteInputsFc02.xExecute				:= tonDelay.Q;
(* Read Holding Registers *)                		
ELSIF _byMbFunction = 03 THEN                   	
	fbReadHoldingRegistersFc03.udiReplyTimeout		:= TO_UDINT(tTimeOut) * 1000; 
	fbReadHoldingRegistersFc03.udiTimeOut			:= TO_UDINT(tTimeOut) * 1000 * 2;
	fbReadHoldingRegistersFc03.uiUnitId				:= usiNodeId;          	
	fbReadHoldingRegistersFc03.uiStartItem			:= TO_UINT(_wMbAdress);
	fbReadHoldingRegistersFc03.pData 				:= _pByte;
	fbReadHoldingRegistersFc03.uiQuantity			:= TO_UINT(_wQuantity);
	fbReadHoldingRegistersFc03.xExecute				:= tonDelay.Q;			
(* Read Input Registers *)	                		
ELSIF _byMbFunction = 04 THEN                   	
	fbReadInputRegistersFc04.udiReplyTimeout		:= TO_UDINT(tTimeOut) * 1000; 
	fbReadInputRegistersFc04.udiTimeOut				:= TO_UDINT(tTimeOut) * 1000 * 2;
	fbReadInputRegistersFc04.uiUnitId				:= usiNodeId;               	
	fbReadInputRegistersFc04.uiStartItem 			:= TO_UINT(_wMbAdress);
	fbReadInputRegistersFc04.pData 					:= _pByte;
	fbReadInputRegistersFc04.uiQuantity				:= TO_UINT(_wQuantity);
	fbReadInputRegistersFc04.xExecute				:= tonDelay.Q;			
(* Write Single Coil *)	                    		
ELSIF _byMbFunction = 05 THEN                   	
	fbWriteSingleCoilFc05.udiReplyTimeout			:= TO_UDINT(tTimeOut) * 1000; 
	fbWriteSingleCoilFc05.udiTimeOut				:= TO_UDINT(tTimeOut) * 1000 * 2;
	fbWriteSingleCoilFc05.uiUnitId					:= usiNodeId;            	
	fbWriteSingleCoilFc05.uiItem 					:= TO_UINT(_wMbAdress);
	fbWriteSingleCoilFc05.xValue 					:= FcBytePointToBoolValue(_pByte);
	fbWriteSingleCoilFc05.xExecute					:= tonDelay.Q;		
(* Write Single Register *)                 		
ELSIF _byMbFunction = 06 THEN                   	
	fbWriteSingleRegisterFc06.udiReplyTimeout		:= TO_UDINT(tTimeOut) * 1000;    
	fbWriteSingleRegisterFc06.udiTimeOut			:= TO_UDINT(tTimeOut) * 1000 * 2; 
	fbWriteSingleRegisterFc06.uiUnitId				:= usiNodeId;           	
	fbWriteSingleRegisterFc06.uiItem	  			:= TO_UINT(_wMbAdress);
	fbWriteSingleRegisterFc06.uiValue 				:= FcBytePointToWordValue(_pByte);
	fbWriteSingleRegisterFc06.xExecute				:= tonDelay.Q;		
(* Write Multiple Coils *)		            		
ELSIF _byMbFunction = 15 THEN                   	
	fbWriteMultipleCoilsFc15.udiReplyTimeout		:= TO_UDINT(tTimeOut) * 1000;
	fbWriteMultipleCoilsFc15.udiTimeOut				:= TO_UDINT(tTimeOut) * 1000 * 2;
	fbWriteMultipleCoilsFc15.uiUnitId				:= usiNodeId;              	
	fbWriteMultipleCoilsFc15.uiStartItem 			:= TO_UINT(_wMbAdress);
	fbWriteMultipleCoilsFc15.pData 					:= _pByte;
	fbWriteMultipleCoilsFc15.uiQuantity				:= TO_UINT(_wQuantity);
	fbWriteMultipleCoilsFc15.xExecute				:= tonDelay.Q;
(* Write Multiple Registers *)                  	
ELSIF _byMbFunction = 16 THEN                   	
	fbWriteMultipleRegistersFc16.udiReplyTimeout	:= TO_UDINT(tTimeOut) * 1000; 
	fbWriteMultipleRegistersFc16.udiTimeOut			:= TO_UDINT(tTimeOut) * 1000 * 2;
	fbWriteMultipleRegistersFc16.uiUnitId			:= usiNodeId;    
	fbWriteMultipleRegistersFc16.uiStartItem 		:= TO_UINT(_wMbAdress);
	fbWriteMultipleRegistersFc16.pData 				:= _pByte;
	fbWriteMultipleRegistersFc16.uiQuantity			:= TO_UINT(_wQuantity);
	fbWriteMultipleRegistersFc16.xExecute			:= tonDelay.Q;	
END_IF;
END_ACTION

ACTION actGetError:
(* Client Error *)
IF _TEMP_MBU_CLIENT_TCP.ClientTcp.xError THEN
	xErrorHappen 	:= _TEMP_MBU_CLIENT_TCP.ClientTcp.xError;
	eErrorID		:= _TEMP_MBU_CLIENT_TCP.ClientTcp.eErrorID;
	eExeptionCode	:= ModbusFB.ExceptionCodes.ACKNOWLEDGE;
	xAbort			:= TRUE;
END_IF;
(* Read Coils Fc01 Error *)
IF fbReadCoilsFc01.xError AND NOT xErrorHappen THEN
	xErrorHappen 	:= fbReadCoilsFc01.xError;
	eErrorID		:= fbReadCoilsFc01.eErrorID;
	eExeptionCode	:= fbReadCoilsFc01.eException;
	xAbort			:= TRUE;
END_IF;
(* Read Discrete Inputs Fc02 Error *)
IF fbReadDiscreteInputsFc02.xError AND NOT xErrorHappen THEN
	xErrorHappen 	:= fbReadDiscreteInputsFc02.xError;
	eErrorID		:= fbReadDiscreteInputsFc02.eErrorID;
	eExeptionCode	:= fbReadDiscreteInputsFc02.eException;
	xAbort			:= TRUE;
END_IF;
(* Read Holding Registers Fc03 Error *)
IF fbReadHoldingRegistersFc03.xError AND NOT xErrorHappen THEN
	xErrorHappen 	:= fbReadHoldingRegistersFc03.xError;
	eErrorID		:= fbReadHoldingRegistersFc03.eErrorID;
	eExeptionCode	:= fbReadHoldingRegistersFc03.eException;
	xAbort			:= TRUE;
END_IF;
(* Read Input Registers Fc04 Error *)
IF fbReadInputRegistersFc04.xError AND NOT xErrorHappen THEN
	xErrorHappen 	:= fbReadInputRegistersFc04.xError;
	eErrorID		:= fbReadInputRegistersFc04.eErrorID;
	eExeptionCode	:= fbReadInputRegistersFc04.eException;
	xAbort			:= TRUE;
END_IF;
(* Write Single Coil Fc05 Error *)
IF fbWriteSingleCoilFc05.xError AND NOT xErrorHappen THEN
	xErrorHappen 	:= fbWriteSingleCoilFc05.xError;
	eErrorID		:= fbWriteSingleCoilFc05.eErrorID;
	eExeptionCode	:= fbWriteSingleCoilFc05.eException;
	xAbort			:= TRUE;
END_IF;
(* Write Single Register Fc06 Error *)
IF fbWriteSingleRegisterFc06.xError AND NOT xErrorHappen THEN
	xErrorHappen 	:= fbWriteSingleRegisterFc06.xError;
	eErrorID		:= fbWriteSingleRegisterFc06.eErrorID;
	eExeptionCode	:= fbWriteSingleRegisterFc06.eException;
	xAbort			:= TRUE;
END_IF;		
(* Write Multiple Coils Fc15 Error *)
IF fbWriteMultipleCoilsFc15.xError AND NOT xErrorHappen THEN
	xErrorHappen 	:= fbWriteMultipleCoilsFc15.xError;
	eErrorID		:= fbWriteMultipleCoilsFc15.eErrorID;
	eExeptionCode	:= fbWriteMultipleCoilsFc15.eException;
	xAbort			:= TRUE;
END_IF;
(* Write Multiple Registers Fc16 Error *)
IF fbWriteMultipleRegistersFc16.xError AND NOT xErrorHappen THEN
	xErrorHappen 	:= fbWriteMultipleRegistersFc16.xError;
	eErrorID		:= fbWriteMultipleRegistersFc16.eErrorID;
	eExeptionCode	:= fbWriteMultipleRegistersFc16.eException;
	xAbort			:= TRUE;
END_IF;
END_ACTION

END_FUNCTION_BLOCK

// 30 Program Organization Units/CLIENTMANAGER/BASE/FB_MB_CLIENTMANAGER
{attribute 'no_assign'}
FUNCTION_BLOCK FB_MB_CLIENTMANAGER EXTENDS CtaAppBmk.fbBMK IMPLEMENTS ITF_MB_CLIENTMANAGER
VAR_OUTPUT
END_VAR
VAR
	_BASE_MBU_CLIENT					:	ITF_CLIENT;
	_TEMP_REG_CLIENT					:	ITF_CLIENT;
	_TEMP_MBU_CLIENT					:	ITF_CLIENT;		
	_COUNT								:	UINT;
	
	xIsWorking							:	BOOL;
	xTrig								:	BOOL;
	xAbort								:	BOOL;
	xErrorHappen						:	BOOL;
	eErrorID							:	ModbusFB.Error;
	eExeptionCode						:	ModbusFB.ExceptionCodes;
	
	usiNodeId							:	USINT;
	
	tTimeOut							:	TIME;
	tReadDelay							:	TIME;
	tWriteDelay							:	TIME;
	tonDelay							:	Standard.TON;
	_byMbFunction						:	BYTE;
	_wMbAdress							:	WORD;
	_pByte								:	POINTER TO BYTE;
	_wQuantity							:	WORD;	
	                					
	fbTimeStop							:	CtaAppTime.fbTimeMeasurement;
	ltTime								:	LTIME;

	_ayITF_MBCLIENT_VIS					:	ARRAY[0..9] OF ITF_CLIENT;

END_VAR

METHOD RELOAD_ARRAY
VAR_INPUT
	xInit	: BOOL;
	xLoadNext10	: BOOL;
	xLoadLast10	: BOOL;
END_VAR
VAR
	diFor				:	DINT;
	ITF_TEMP_CLIENT_VIS	:	ITF_CLIENT;
	ITF_TEMP_SAFE		:	ITF_CLIENT;
	ITF_TEMP_LAST_VALID	:	ITF_CLIENT;
END_VAR
(* Init Array *)
IF xInit THEN
	_ayITF_MBCLIENT_VIS[LOWER_BOUND(_ayITF_MBCLIENT_VIS,1)] := _BASE_MBU_CLIENT;
	FOR diFor := LOWER_BOUND(_ayITF_MBCLIENT_VIS,1) TO UPPER_BOUND(_ayITF_MBCLIENT_VIS,1) -1 DO
		IF __QUERYINTERFACE(_ayITF_MBCLIENT_VIS[diFor],ITF_TEMP_CLIENT_VIS) THEN
			_ayITF_MBCLIENT_VIS[diFor + 1]	:= _ayITF_MBCLIENT_VIS[diFor].LOW_SYBIL;
		ELSE
			_ayITF_MBCLIENT_VIS[diFor + 1] := 0;
		END_IF;	
	END_FOR;
(* Load Next 10 *)
ELSIF xLoadNext10 THEN
	IF __QUERYINTERFACE(_ayITF_MBCLIENT_VIS[UPPER_BOUND(_ayITF_MBCLIENT_VIS,1)],ITF_TEMP_CLIENT_VIS) THEN
		_ayITF_MBCLIENT_VIS[LOWER_BOUND(_ayITF_MBCLIENT_VIS,1)] := ITF_TEMP_CLIENT_VIS.LOW_SYBIL;
		FOR diFor := LOWER_BOUND(_ayITF_MBCLIENT_VIS,1) TO UPPER_BOUND(_ayITF_MBCLIENT_VIS,1) -1 DO
			IF __QUERYINTERFACE(_ayITF_MBCLIENT_VIS[diFor],ITF_TEMP_CLIENT_VIS) THEN
				_ayITF_MBCLIENT_VIS[diFor + 1]	:= _ayITF_MBCLIENT_VIS[diFor].LOW_SYBIL;
			ELSE
				_ayITF_MBCLIENT_VIS[diFor + 1] := 0;
			END_IF;	
		END_FOR;
	END_IF;
(* Load Last 10 *)
ELSIF xLoadLast10 THEN
	IF __QUERYINTERFACE(_ayITF_MBCLIENT_VIS[LOWER_BOUND(_ayITF_MBCLIENT_VIS,1)],ITF_TEMP_CLIENT_VIS) THEN
		IF __QUERYINTERFACE(_ayITF_MBCLIENT_VIS[LOWER_BOUND(_ayITF_MBCLIENT_VIS,1)].BIG_SYBIL,ITF_TEMP_SAFE) THEN
			_ayITF_MBCLIENT_VIS[UPPER_BOUND(_ayITF_MBCLIENT_VIS,1)] := ITF_TEMP_CLIENT_VIS.BIG_SYBIL;
			FOR diFor := UPPER_BOUND(_ayITF_MBCLIENT_VIS,1) TO LOWER_BOUND(_ayITF_MBCLIENT_VIS,1) + 1 BY -1 DO 
				IF __QUERYINTERFACE(_ayITF_MBCLIENT_VIS[diFor],ITF_TEMP_CLIENT_VIS) THEN
					ITF_TEMP_LAST_VALID  			:= _ayITF_MBCLIENT_VIS[diFor];
					_ayITF_MBCLIENT_VIS[diFor - 1]	:= _ayITF_MBCLIENT_VIS[diFor].BIG_SYBIL;
				ELSE
					(* Resort if new ones Inside *)
					_ayITF_MBCLIENT_VIS[LOWER_BOUND(_ayITF_MBCLIENT_VIS,1)] := ITF_TEMP_LAST_VALID;
					FOR diFor := LOWER_BOUND(_ayITF_MBCLIENT_VIS,1) TO UPPER_BOUND(_ayITF_MBCLIENT_VIS,1) -1 DO
						IF __QUERYINTERFACE(_ayITF_MBCLIENT_VIS[diFor],ITF_TEMP_CLIENT_VIS) THEN
							_ayITF_MBCLIENT_VIS[diFor + 1]	:= _ayITF_MBCLIENT_VIS[diFor].LOW_SYBIL;
						ELSE
							_ayITF_MBCLIENT_VIS[diFor + 1] := 0;
						END_IF;	
					END_FOR;					
				END_IF;	
			END_FOR;
		END_IF;
	END_IF;	
END_IF;
END_METHOD

METHOD ADD_MODBUS_CLIENT
VAR_INPUT
	ITF_CLIENT_IN	:	ITF_CLIENT;
END_VAR
IF NOT CHECK_IF_EXIST(ITF_CLIENT_IN) THEN
	IF __QUERYINTERFACE(ITF_CLIENT_IN,ITF_CLIENT_IN) THEN
		IF __QUERYINTERFACE(_BASE_MBU_CLIENT,_BASE_MBU_CLIENT) THEN
			IF __QUERYINTERFACE(_TEMP_REG_CLIENT,_TEMP_REG_CLIENT) THEN
				_TEMP_REG_CLIENT.LOW_SYBIL := ITF_CLIENT_IN;
				_TEMP_REG_CLIENT := ITF_CLIENT_IN;
			ELSE
				_BASE_MBU_CLIENT.LOW_SYBIL := ITF_CLIENT_IN;
				_TEMP_REG_CLIENT := ITF_CLIENT_IN;		
			END_IF;		
		ELSE
			_BASE_MBU_CLIENT := ITF_CLIENT_IN;
		END_IF;
		THIS^.RELOAD_ARRAY(TRUE,FALSE,FALSE);
		_COUNT := _COUNT + 1;
	END_IF;
END_IF;
END_METHOD

METHOD CHECK_IF_EXIST : BOOL
VAR_INPUT
	ITF_CLIENT_IN	:	ITF_CLIENT;
END_VAR
VAR
	ITF_CLIENT_TEMP	:	ITF_CLIENT;
END_VAR
IF __QUERYINTERFACE(_BASE_MBU_CLIENT,ITF_CLIENT_TEMP) THEN
	REPEAT
		IF __QUERYINTERFACE(ITF_CLIENT_TEMP,ITF_CLIENT_TEMP) THEN
			IF ITF_CLIENT_IN = ITF_CLIENT_TEMP THEN
				CHECK_IF_EXIST := TRUE;
			END_IF
			ITF_CLIENT_TEMP := ITF_CLIENT_TEMP.LOW_SYBIL;
		ELSE
			ITF_CLIENT_TEMP := 0;
		END_IF;
	UNTIL ITF_CLIENT_TEMP = 0 OR CHECK_IF_EXIST 
	END_REPEAT;
END_IF
END_METHOD

PROPERTY AY_ITF_MBCLIENT_VIS : ARRAY [0..9] OF ITF_CLIENT
GET
AY_ITF_MBCLIENT_VIS := _ayITF_MBCLIENT_VIS;
END_GET
END_PROPERTY

PROPERTY ITF_BASE_CLIENT : ITF_CLIENT
GET
END_GET
END_PROPERTY

PROPERTY OperationTime : LTIME
GET
OperationTime := ltTime;
END_GET
END_PROPERTY

METHOD INTERNAL COUNT_ENABLED : UINT
VAR
	ITF_CLIENT_TEMP	:	ITF_CLIENT;
END_VAR
IF __QUERYINTERFACE(_BASE_MBU_CLIENT,ITF_CLIENT_TEMP) THEN
	REPEAT
		IF __QUERYINTERFACE(ITF_CLIENT_TEMP,ITF_CLIENT_TEMP) THEN
			IF ITF_CLIENT_TEMP.ENABLE THEN
				COUNT_ENABLED := COUNT_ENABLED + 1;
			END_IF
			ITF_CLIENT_TEMP := ITF_CLIENT_TEMP.LOW_SYBIL;
		ELSE
			ITF_CLIENT_TEMP := 0;
		END_IF;
	UNTIL ITF_CLIENT_TEMP = 0
	END_REPEAT;
END_IF
END_METHOD

END_FUNCTION_BLOCK

// 21 Interface/CLIENTMANAGER/TCP/ITF_MB_CLIENTMANAGER_TCP
INTERFACE ITF_MB_CLIENTMANAGER_TCP EXTENDS ITF_MB_CLIENTMANAGER

END_INTERFACE

// 30 Program Organization Units/FC/FcBytePointToBoolValue
FUNCTION FcBytePointToBoolValue : BOOL
VAR_INPUT
	_pByte			:	POINTER TO BYTE;
END_VAR
VAR
	_pBool			:	POINTER TO BOOL;
END_VAR

IF _pByte <> 0 THEN
	_pBool := _pByte;
	FcBytePointToBoolValue := _pBool^;
END_IF;

END_FUNCTION

// 30 Program Organization Units/FC/FcBytePointToWordValue
FUNCTION FcBytePointToWordValue : WORD
VAR_INPUT
	_pByte			:	POINTER TO BYTE;
END_VAR
VAR
	_pWord			:	POINTER TO Word;
END_VAR

IF _pByte <> 0 THEN
	_pWord := _pByte;
	FcBytePointToWordValue := _pWord^;
END_IF;

END_FUNCTION

// 30 Program Organization Units/SERVER/FB_SERVER
{attribute 'no_assign'}
FUNCTION_BLOCK FB_SERVER IMPLEMENTS ITF_SERVER_INFO_PARA
VAR_INPUT
END_VAR
VAR_OUTPUT
	xTimeOutTcpWatchDog				:	BOOL;
	xTimeOutSerialWatchDog			:	BOOL;
END_VAR
VAR
	(* Servers *)	
	fbServerTcp						:	ServerTCP_Extended		:= (udiLogOptions			:= ModbusFB.LoggingOptions.All);
	fbServerSerial					:	ServerSerial_Extended	:= (udiLogOptions			:= ModbusFB.LoggingOptions.All);
	
	(* Data *)
    ayxCoil                         :   ARRAY[0..16#FFFF] OF BOOL;
    ayxDiscretInput                 :   ARRAY[0..16#FFFF] OF BOOL;  
    aywInputRegister                :   ARRAY[0..16#FFFF] OF WORD;
    aywHoldingRegister              :   ARRAY[0..16#FFFF] OF WORD; 	
	
	(* Data Model *)
	scDataModel						:	ModbusFB.TableDefinitions;
	scSectionCoil					:	ARRAY[0..1] OF ModbusFB.TableSection;
	scSectionDiscretInput			:	ARRAY[0..1] OF ModbusFB.TableSection;
	scSectionInputRegister			:	ARRAY[0..1] OF ModbusFB.TableSection;
	scSectionHoldingRegister		:	ARRAY[0..1] OF ModbusFB.TableSection;
	
	(* Help Variable *)
	xEnableTcp						:	BOOL;
	xEnableSerial					:	BOOL;
	scRequestDataTcp				:	Modbusfb.RequestData;
	scRequestDataSerial				:	Modbusfb.RequestData;
	fbNoTcpAccesSince				:	CtaAppTime.fbTimeMeasurement;	
	tNoTcpAccesSince				:	TIME;
	fbNoSerialAccesSince			:	CtaAppTime.fbTimeMeasurement;	
	tNoSerialAccesSince				:	TIME;
	
	(* Config *)
	fbConfigFile					:	CtaSysConfig.fbConfigFile;
	scParameter						:	scModBusServerParameter;
END_VAR

(* Config *)
actConfig();

(* DataModell *)
actDataModel();

(* TCP Server *)
actTcp();

(* Serial Server *)
actSerial();

ACTION actConfig:
(* Config File *)
fbConfigFile();

scParameter.scSerial.fbxEnable              (_usiParaNr :=  1, ItfConfigFb := fbConfigFile                                              );
scParameter.scSerial.fbenPort				(_usiParaNr :=  2, ItfConfigFb := fbConfigFile , _MinInit :=    0     , _MaxInit :=     10	);
scParameter.scSerial.fbusiNodeId            (_usiParaNr :=  3, ItfConfigFb := fbConfigFile , _MinInit :=    0     , _MaxInit :=     247 ); 
scParameter.scSerial.fbdwBaudrate           (_usiParaNr :=  4, ItfConfigFb := fbConfigFile , _MinInit := 9600     , _MaxInit :=   115200);
scParameter.scSerial.fbbyDataBits           (_usiParaNr :=  5, ItfConfigFb := fbConfigFile , _MinInit :=    5     , _MaxInit :=       8 );
scParameter.scSerial.fbenParity             (_usiParaNr :=  6, ItfConfigFb := fbConfigFile , _MinInit :=    0     , _MaxInit :=       5 );
scParameter.scSerial.fbenStopBits           (_usiParaNr :=  7, ItfConfigFb := fbConfigFile , _MinInit :=    0     , _MaxInit :=       5 );
scParameter.scSerial.fbenDTRControl         (_usiParaNr :=  8, ItfConfigFb := fbConfigFile , _MinInit :=    0     , _MaxInit :=       2 );
scParameter.scSerial.fbenRTSControl         (_usiParaNr :=  9, ItfConfigFb := fbConfigFile , _MinInit :=    0     , _MaxInit :=       2 );
scParameter.scSerial.fbxRtuAscii            (_usiParaNr := 10, ItfConfigFb := fbConfigFile                                              );
scParameter.scSerial.fbxEnableWatchDog      (_usiParaNr := 11, ItfConfigFb := fbConfigFile                                              );
scParameter.scSerial.fbtWatchDog            (_usiParaNr := 12, ItfConfigFb := fbConfigFile , _MinInit := T#1S     , _MaxInit :=   T#30M );
scParameter.scTcp.fbxEnable                 (_usiParaNr := 13, ItfConfigFb := fbConfigFile                                              );
scParameter.scTcp.fbwPort                   (_usiParaNr := 14, ItfConfigFb := fbConfigFile , _MinInit :=    0     , _MaxInit := 16#FFFF );
scParameter.scTcp.fbxEnableWatchDog         (_usiParaNr := 15, ItfConfigFb := fbConfigFile                                              );
scParameter.scTcp.fbtWatchDog               (_usiParaNr := 16, ItfConfigFb := fbConfigFile , _MinInit := T#50MS   , _MaxInit :=   T#30M );
scParameter.scTcp.fbstInterface				(_usiParaNr := 17, ItfConfigFb := fbConfigFile 												);
scParameter.loggingOp						(_usiParaNr := 18, ItfConfigFb := fbConfigFile,	_WertInit := TO_WORD(ModbusFB.LoggingOptions.Internals)	);




(* Serial Change reset enable*)
IF scParameter.scSerial.fbxEnable.proStateChanged         	OR
   scParameter.scSerial.fbenPort.proStateChanged			OR
   scParameter.scSerial.fbusiNodeId.proStateChanged       	OR
   scParameter.scSerial.fbdwBaudrate.proStateChanged      	OR 
   scParameter.scSerial.fbbyDataBits.proStateChanged      	OR 
   scParameter.scSerial.fbenParity.proStateChanged       	OR 
   scParameter.scSerial.fbenStopBits.proStateChanged     	OR 
   scParameter.scSerial.fbenDTRControl.proStateChanged    	OR 
   scParameter.scSerial.fbenRTSControl.proStateChanged    	OR 
   scParameter.scSerial.fbxRtuAscii.proStateChanged      	OR 
   scParameter.scSerial.fbxEnableWatchDog.proStateChanged 	OR 
   scParameter.scSerial.fbtWatchDog.proStateChanged       	THEN
	xEnableSerial := FALSE;
ELSE
	xEnableSerial := scParameter.scSerial.fbxEnable.proValue;
END_IF;

(* Tcp Change reset enable*)
IF scParameter.scTcp.fbxEnable.proStateChanged				OR     
   scParameter.scTcp.fbwPort.proStateChanged				OR                                
   scParameter.scTcp.fbxEnableWatchDog.proStateChanged		OR  
   scParameter.scTcp.fbtWatchDog.proStateChanged			OR  
   scParameter.scTcp.fbstInterface.proStateChanged			THEN	
	xEnableTcp := FALSE;
ELSE
	xEnableTcp := scParameter.scTcp.fbxEnable.proValue;
END_IF;
END_ACTION

ACTION actDataModel:
(* Coil Data Model *)
scSectionCoil[0].pStartAddr						:= ADR(ayxCoil[0]);
scSectionCoil[0].uiStart						:= 0;
scSectionCoil[0].uiNumDataItems					:= 16#0001;
scSectionCoil[0].uiDataItemSize					:= 1;
scSectionCoil[1].pStartAddr						:= ADR(ayxCoil[1]);
scSectionCoil[1].uiStart						:= 1;
scSectionCoil[1].uiNumDataItems					:= 16#FFFF;
scSectionCoil[1].uiDataItemSize					:= 1;

scDataModel.tableCoils.pSections 				:= ADR(scSectionCoil);
scDataModel.tableCoils.uiNumSections			:= 2;

(* Discret Input Data Model *)
scSectionDiscretInput[0].pStartAddr				:= ADR(ayxDiscretInput[0]);
scSectionDiscretInput[0].uiStart				:= 0;
scSectionDiscretInput[0].uiNumDataItems			:= 16#0001;
scSectionDiscretInput[0].uiDataItemSize			:= 1;
scSectionDiscretInput[1].pStartAddr				:= ADR(ayxDiscretInput[1]);
scSectionDiscretInput[1].uiStart				:= 1;
scSectionDiscretInput[1].uiNumDataItems			:= 16#FFFF;
scSectionDiscretInput[1].uiDataItemSize			:= 1;

scDataModel.tableDiscreteInputs.pSections		:= ADR(scSectionDiscretInput);
scDataModel.tableDiscreteInputs.uiNumSections	:= 2;

(* Holding Register Data Model *)
scSectionHoldingRegister[0].pStartAddr			:= ADR(aywHoldingRegister[0]);
scSectionHoldingRegister[0].uiStart				:= 0;
scSectionHoldingRegister[0].uiNumDataItems		:= 16#0001;
scSectionHoldingRegister[0].uiDataItemSize		:= 16;
scSectionHoldingRegister[1].pStartAddr			:= ADR(aywHoldingRegister[1]);
scSectionHoldingRegister[1].uiStart				:= 1;
scSectionHoldingRegister[1].uiNumDataItems		:= 16#FFFF;
scSectionHoldingRegister[1].uiDataItemSize		:= 16;

scDataModel.tableHoldingRegisters.pSections		:= ADR(scSectionHoldingRegister);
scDataModel.tableHoldingRegisters.uiNumSections := 2;

(* Input Register Data Model *)
scSectionInputRegister[0].pStartAddr			:= ADR(aywInputRegister[0]);
scSectionInputRegister[0].uiStart				:= 0;
scSectionInputRegister[0].uiNumDataItems		:= 16#0001;
scSectionInputRegister[0].uiDataItemSize		:= 16;
scSectionInputRegister[1].pStartAddr			:= ADR(aywInputRegister[1]);
scSectionInputRegister[1].uiStart				:= 1;
scSectionInputRegister[1].uiNumDataItems		:= 16#FFFF;
scSectionInputRegister[1].uiDataItemSize		:= 16;

scDataModel.tableInputRegisters.pSections		:= ADR(scSectionInputRegister);
scDataModel.tableInputRegisters.uiNumSections	:= 2;
END_ACTION

ACTION actSerial:
(* Serial Server *)
fbServerSerial(	xEnable	 				:= xEnableSerial,
				dataModel 				:= scDataModel,
				tInactivityInfoTime		:= TO_UDINT(T#30S),
				uiUnitId				:= TO_UINT(scParameter.scSerial.fbusiNodeId.proValue),
				iPort					:= scParameter.scSerial.fbenPort.proValue,
				dwBaudrate				:= scParameter.scSerial.fbdwBaudrate.proValue,
				byDataBits				:= scParameter.scSerial.fbbyDataBits.proValue,
				eParity					:= scParameter.scSerial.fbenParity.proValue,
				eStopBits				:= scParameter.scSerial.fbenStopBits.proValue,
				eDTRcontrol				:= scParameter.scSerial.fbenDTRControl.proValue,
				eRTScontrol				:= scParameter.scSerial.fbenRTSControl.proValue,
				eRtuAscii				:= SEL(scParameter.scSerial.fbxRtuAscii.proValue,ModbusFB.RtuAscii.RTU,ModbusFB.RtuAscii.ASCII),
				udiLogOptions			:= scParameter.loggingOp.proValue);

(* Last Acces Time and WatchDog Timeout*)
IF xEnableSerial THEN	
	(* Get Last Acces *)
	IF fbServerSerial.xWriteRequest OR fbServerSerial.xReadRequest THEN
		fbNoSerialAccesSince.Start();
		tNoSerialAccesSince := T#0MS;
	ELSE
		tNoSerialAccesSince := TO_TIME(fbNoSerialAccesSince.Stop());
	END_IF;
	(* WatchDog Timeout *)
	IF scParameter.scSerial.fbxEnableWatchDog.xValue THEN
		IF scParameter.scSerial.fbtWatchDog.tValue < tNoSerialAccesSince THEN
			xTimeOutSerialWatchDog := TRUE;
		ELSE
			xTimeOutSerialWatchDog := FALSE;
		END_IF;
	ELSE
		xTimeOutSerialWatchDog := FALSE;
	END_IF;	
ELSE
	fbNoSerialAccesSince.Start();
	tNoSerialAccesSince := T#0MS;	
	xTimeOutSerialWatchDog := FALSE;
END_IF;
		
(* Requestdata Serial *)				
scRequestDataSerial := fbServerSerial.RequestData;
END_ACTION

ACTION actTcp:
(* TCP Server *)
fbServerTcp(	xEnable	 				:= xEnableTcp,
				dataModel 				:= scDataModel,
				tInactivityInfoTime		:= 0,
				wsInterfaceName			:= TO_WSTRING(scParameter.scTcp.fbstInterface.proValue),
				uiPort					:= TO_UINT(scParameter.scTcp.fbwPort.proValue),
				xReset					:= fbServerTcp.xError,
				udiLogOptions			:= scParameter.loggingOp.proValue);

(* Last Acces Time and WatchDog Timeout*)
IF xEnableTcp THEN	
	(* Get Last Acces *)
	IF fbServerTcp.xWriteRequest OR fbServerTcp.xReadRequest THEN
		fbNoTcpAccesSince.Start();
		tNoTcpAccesSince := T#0MS;
	ELSE
		tNoTcpAccesSince := TO_TIME(fbNoTcpAccesSince.Stop());
	END_IF;
	(* WatchDog Timeout *)
	IF scParameter.scTcp.fbxEnableWatchDog.xValue THEN
		IF scParameter.scTcp.fbtWatchDog.tValue < tNoTcpAccesSince THEN
			xTimeOutTcpWatchDog := TRUE;
		ELSE
			xTimeOutTcpWatchDog := FALSE;
		END_IF;
	ELSE
		xTimeOutTcpWatchDog := FALSE;
	END_IF;	
ELSE
	fbNoTcpAccesSince.Start();
	tNoTcpAccesSince := T#0MS;	
	xTimeOutTcpWatchDog := FALSE;
END_IF;
			
(* Requestdata TCP *)		
scRequestDataTcp := fbServerTcp.RequestData;
END_ACTION

METHOD metGetCoil : BOOL
VAR_INPUT
	wAdr	: WORD;
END_VAR
IF wAdr >= 0 AND wAdr <= 16#FFFF THEN
	metGetCoil := ayxCoil[wAdr];
END_IF;
END_METHOD

METHOD metGetHoldingRegister : WORD
VAR_INPUT
	wAdr	: WORD;
END_VAR
IF wAdr >= 0 AND wAdr <= 16#FFFF THEN
	metGetHoldingRegister := aywHoldingRegister[wAdr];
END_IF;
END_METHOD

METHOD metSetCoil : BOOL
VAR_INPUT
	wAdr	: WORD;
	xValue	: BOOL;
END_VAR
IF wAdr >= 0 AND wAdr <= 16#FFFF THEN
	ayxCoil[wAdr] := xValue ;
	metSetCoil := TRUE;
END_IF;
END_METHOD

METHOD metSetDiscretInput : BOOL
VAR_INPUT
	wAdr	: WORD;
	xValue	: BOOL;
END_VAR
IF wAdr >= 0 AND wAdr <= 16#FFFF THEN
	ayxDiscretInput[wAdr] := xValue ;
	metSetDiscretInput := TRUE;
END_IF;
END_METHOD

METHOD metSetHoldingRegister : BOOL
VAR_INPUT
	wAdr	: WORD;
	wValue	: WORD;
END_VAR
IF wAdr >= 0 AND wAdr <= 16#FFFF THEN
	aywHoldingRegister[wAdr] := wValue ;
	metSetHoldingRegister := TRUE;
END_IF;
END_METHOD

METHOD metSetInputRegister : BOOL
VAR_INPUT
	wAdr	: WORD;
	wValue	: WORD;
END_VAR
IF wAdr >= 0 AND wAdr <= 16#FFFF THEN
	aywInputRegister[wAdr] := wValue ;
	metSetInputRegister := TRUE;
END_IF;
END_METHOD

PROPERTY P_Serial_fbxEnableWatchDog : CtaSysConfig.ITF_BOOL
GET
P_Serial_fbxEnableWatchDog := scParameter.scSerial.fbxEnableWatchDog;
END_GET
END_PROPERTY

PROPERTY P_Serial_fbxRtuAscii : CtaSysConfig.ITF_BOOL
GET
P_Serial_fbxRtuAscii := scParameter.scSerial.fbxRtuAscii;
END_GET
END_PROPERTY

PROPERTY NoSerialAccesSince : TIME
GET
NoSerialAccesSince := tNoSerialAccesSince;
END_GET
END_PROPERTY

PROPERTY P_Serial_fbbyDataBits : CtaSysConfig.ITF_BYTE
GET
P_Serial_fbbyDataBits := scParameter.scSerial.fbbyDataBits;
END_GET
END_PROPERTY

PROPERTY P_Serial_fbdwBaudrate : CtaSysConfig.ITF_DWORD
GET
P_Serial_fbdwBaudrate := scParameter.scSerial.fbdwBaudrate;
END_GET
END_PROPERTY

PROPERTY P_Serial_fbenDTRControl : CtaSysConfig.ITF_BYTE
GET
P_Serial_fbenDTRControl := scParameter.scSerial.fbenDTRControl;
END_GET
END_PROPERTY

PROPERTY P_Serial_fbenParity : CtaSysConfig.ITF_BYTE
GET
P_Serial_fbenParity := scParameter.scSerial.fbenParity;
END_GET
END_PROPERTY

PROPERTY P_Serial_fbenPort : CtaSysConfig.ITF_INT
GET
P_Serial_fbenPort := scParameter.scSerial.fbenPort;
END_GET
END_PROPERTY

PROPERTY P_Serial_fbenRTSControl : CtaSysConfig.ITF_BYTE
GET
P_Serial_fbenRTSControl := scParameter.scSerial.fbenRTSControl;
END_GET
END_PROPERTY

PROPERTY P_Serial_fbenStopBits : CtaSysConfig.ITF_BYTE
GET
P_Serial_fbenStopBits := scParameter.scSerial.fbenStopBits;
END_GET
END_PROPERTY

PROPERTY P_Serial_fbtWatchDog : CtaSysConfig.ITF_TIME
GET
P_Serial_fbtWatchDog := scParameter.scSerial.fbtWatchDog;
END_GET
END_PROPERTY

PROPERTY P_Serial_fbusiNodeId : CtaSysConfig.ITF_USINT
GET
P_Serial_fbusiNodeId := scParameter.scSerial.fbusiNodeId;
END_GET
END_PROPERTY

PROPERTY P_Serial_fbxEnable : CtaSysConfig.ITF_BOOL
GET
P_Serial_fbxEnable := scParameter.scSerial.fbxEnable;
END_GET
END_PROPERTY

PROPERTY RequestDataSerial : String
GET
(* Read Requests *)
IF 		scRequestDataSerial.fc =  1 OR
		scRequestDataSerial.fc =  2 OR
		scRequestDataSerial.fc =  3 OR
		scRequestDataSerial.fc =  4 THEN
		RequestDataSerial := 	CONCAT('FC: ',
							CONCAT(TO_STRING(scRequestDataSerial.fc),
							CONCAT('$NADR R: ',
							CONCAT(TO_STRING(scRequestDataSerial.u.read.uiStartAddress),
							CONCAT('$NTO: ',TO_STRING(scRequestDataSerial.u.read.uiStartAddress + scRequestDataSerial.u.read.uiQuantity -1))))));
							
(* Write Single Requests *)
ELSIF	scRequestDataSerial.fc =  5 OR
		scRequestDataSerial.fc =  6 THEN
		RequestDataSerial := 	CONCAT('FC: ',
							CONCAT(TO_STRING(scRequestDataSerial.fc),
							CONCAT('$NADR W: ',TO_STRING(scRequestDataSerial.u.writeSingle.uiAddress))));
							
(* Read Exeption State and Diagnostic*)
ELSIF	scRequestDataSerial.fc =  7 OR
		scRequestDataSerial.fc =  8 OR
		scRequestDataSerial.fc = 11 OR
		scRequestDataSerial.fc = 12 THEN
		RequestDataSerial := 	CONCAT('FC: ',
							CONCAT(TO_STRING(scRequestDataSerial.fc),
							CONCAT('$NDIA: ',TO_STRING(scRequestDataSerial.u.diagnostics.subFc))));	
							
(* Write Multiple *)
ELSIF 	scRequestDataSerial.fc = 15 OR
		scRequestDataSerial.fc = 16 THEN
		RequestDataSerial := 	CONCAT('FC: ',
							CONCAT(TO_STRING(scRequestDataSerial.fc),
							CONCAT('$NADR W: ',
							CONCAT(TO_STRING(scRequestDataSerial.u.writeMultiple.uiStartAddress),
							CONCAT('$NTO: ',TO_STRING(scRequestDataSerial.u.writeMultiple.uiStartAddress + scRequestDataSerial.u.writeMultiple.uiQuantity-1))))));

(* Report Server ID *)
ELSIF	scRequestDataSerial.fc = 17 THEN
		RequestDataSerial := 	CONCAT('FC: ',
							CONCAT(TO_STRING(scRequestDataSerial.fc),' REPORT SERVER ID'));	
(* Read File Record *)
ELSIF	scRequestDataSerial.fc = 20 THEN
		RequestDataSerial := 	CONCAT('FC: ',
							CONCAT(TO_STRING(scRequestDataSerial.fc),' Read File'));

(* Write File Record *)
ELSIF	scRequestDataSerial.fc = 21 THEN
		RequestDataSerial := 	CONCAT('FC: ',
							CONCAT(TO_STRING(scRequestDataSerial.fc),' Write File'));		

(* Write Mask Register *)
ELSIF 	scRequestDataSerial.fc = 22 THEN
		RequestDataSerial := 	CONCAT('FC: ',
							CONCAT(TO_STRING(scRequestDataSerial.fc),' Mask Write Register'));	

(* Read Write Multiple *)
ELSIF 	scRequestDataSerial.fc = 23 THEN
		RequestDataSerial := 	CONCAT('FC: ',
							CONCAT(TO_STRING(scRequestDataSerial.fc),
							CONCAT('$NADR R: ',
							CONCAT(TO_STRING(scRequestDataSerial.u.readWriteMultipleRegisters.uiReadStartAddress),
							CONCAT('$NTO: ',
							CONCAT(TO_STRING(scRequestDataSerial.u.readWriteMultipleRegisters.uiReadStartAddress + scRequestDataSerial.u.readWriteMultipleRegisters.uiQuantityRead -1), 
							CONCAT('$NADR W: ',
							CONCAT(TO_STRING(scRequestDataSerial.u.readWriteMultipleRegisters.uiWriteStartAddress),
							CONCAT('$NTO: ',TO_STRING(scRequestDataSerial.u.readWriteMultipleRegisters.uiWriteStartAddress + scRequestDataSerial.u.readWriteMultipleRegisters.uiQuantityWrite -1))))))))));

(* Read FIFO *)
ELSIF 	scRequestDataSerial.fc = 24 THEN
		RequestDataSerial := 	CONCAT('FC: ',
							CONCAT(TO_STRING(scRequestDataSerial.fc),' Read FIFO'));	

(* Read ITF *)
ELSIF 	scRequestDataSerial.fc = 43 THEN
		RequestDataSerial := 	CONCAT('FC: ',
							CONCAT(TO_STRING(scRequestDataSerial.fc),' Read ITF'));	

END_IF;
END_GET
END_PROPERTY

PROPERTY TimeOutSerialWatchDog : BOOL
GET
TimeOutSerialWatchDog := xTimeOutSerialWatchDog;
END_GET
END_PROPERTY

PROPERTY TimeOutTcpWatchDog : BOOL
GET
TimeOutTcpWatchDog := xTimeOutTcpWatchDog;
END_GET
END_PROPERTY

PROPERTY P_Tcp_fbwPort : CtaSysConfig.ITF_WORD
GET
P_Tcp_fbwPort := scParameter.scTcp.fbwPort;
END_GET
END_PROPERTY

PROPERTY P_Tcp_fbxEnable : CtaSysConfig.ITF_BOOL
GET
P_Tcp_fbxEnable := scParameter.scTcp.fbxEnable;
END_GET
END_PROPERTY

PROPERTY P_Tcp_fbxEnableWatchDog : CtaSysConfig.ITF_BOOL
GET
P_Tcp_fbxEnableWatchDog := scParameter.scTcp.fbxEnableWatchDog;
END_GET
END_PROPERTY

PROPERTY RequestDataTcp : String
GET
(* Read Requests *)
IF 		scRequestDataTcp.fc =  1 OR
		scRequestDataTcp.fc =  2 OR
		scRequestDataTcp.fc =  3 OR
		scRequestDataTcp.fc =  4 THEN
		RequestDataTcp := 	CONCAT('FC: ',
							CONCAT(TO_STRING(scRequestDataTcp.fc),
							CONCAT('$NADR R: ',
							CONCAT(TO_STRING(scRequestDataTcp.u.read.uiStartAddress),
							CONCAT('$NTO: ',TO_STRING(scRequestDataTcp.u.read.uiStartAddress + scRequestDataTcp.u.read.uiQuantity -1))))));
							
(* Write Single Requests *)
ELSIF	scRequestDataTcp.fc =  5 OR
		scRequestDataTcp.fc =  6 THEN
		RequestDataTcp := 	CONCAT('FC: ',
							CONCAT(TO_STRING(scRequestDataTcp.fc),
							CONCAT('$NADR W: ',TO_STRING(scRequestDataTcp.u.writeSingle.uiAddress))));
							
(* Read Exeption State and Diagnostic*)
ELSIF	scRequestDataTcp.fc =  7 OR
		scRequestDataTcp.fc =  8 OR
		scRequestDataTcp.fc = 11 OR
		scRequestDataTcp.fc = 12 THEN
		RequestDataTcp := 	CONCAT('FC: ',
							CONCAT(TO_STRING(scRequestDataTcp.fc),
							CONCAT('$NDIA: ',TO_STRING(scRequestDataTcp.u.diagnostics.subFc))));	
							
(* Write Multiple *)
ELSIF 	scRequestDataTcp.fc = 15 OR
		scRequestDataTcp.fc = 16 THEN
		RequestDataTcp := 	CONCAT('FC: ',
							CONCAT(TO_STRING(scRequestDataTcp.fc),
							CONCAT('$NADR W: ',
							CONCAT(TO_STRING(scRequestDataTcp.u.writeMultiple.uiStartAddress),
							CONCAT('$NTO: ',TO_STRING(scRequestDataTcp.u.writeMultiple.uiStartAddress + scRequestDataTcp.u.writeMultiple.uiQuantity-1))))));

(* Report Server ID *)
ELSIF	scRequestDataTcp.fc = 17 THEN
		RequestDataTcp := 	CONCAT('FC: ',
							CONCAT(TO_STRING(scRequestDataTcp.fc),' REPORT SERVER ID'));	
(* Read File Record *)
ELSIF	scRequestDataTcp.fc = 20 THEN
		RequestDataTcp := 	CONCAT('FC: ',
							CONCAT(TO_STRING(scRequestDataTcp.fc),' Read File'));

(* Write File Record *)
ELSIF	scRequestDataTcp.fc = 21 THEN
		RequestDataTcp := 	CONCAT('FC: ',
							CONCAT(TO_STRING(scRequestDataTcp.fc),' Write File'));		

(* Write Mask Register *)
ELSIF 	scRequestDataTcp.fc = 22 THEN
		RequestDataTcp := 	CONCAT('FC: ',
							CONCAT(TO_STRING(scRequestDataTcp.fc),' Mask Write Register'));	

(* Read Write Multiple *)
ELSIF 	scRequestDataTcp.fc = 23 THEN
		RequestDataTcp := 	CONCAT('FC: ',
							CONCAT(TO_STRING(scRequestDataTcp.fc),
							CONCAT('$NADR R: ',
							CONCAT(TO_STRING(scRequestDataTcp.u.readWriteMultipleRegisters.uiReadStartAddress),
							CONCAT('$NTO: ',
							CONCAT(TO_STRING(scRequestDataTcp.u.readWriteMultipleRegisters.uiReadStartAddress + scRequestDataTcp.u.readWriteMultipleRegisters.uiQuantityRead -1), 
							CONCAT('$NADR W: ',
							CONCAT(TO_STRING(scRequestDataTcp.u.readWriteMultipleRegisters.uiWriteStartAddress),
							CONCAT('$NTO: ',TO_STRING(scRequestDataTcp.u.readWriteMultipleRegisters.uiWriteStartAddress + scRequestDataTcp.u.readWriteMultipleRegisters.uiQuantityWrite -1))))))))));

(* Read FIFO *)
ELSIF 	scRequestDataTcp.fc = 24 THEN
		RequestDataTcp := 	CONCAT('FC: ',
							CONCAT(TO_STRING(scRequestDataTcp.fc),' Read FIFO'));	

(* Read ITF *)
ELSIF 	scRequestDataTcp.fc = 43 THEN
		RequestDataTcp := 	CONCAT('FC: ',
							CONCAT(TO_STRING(scRequestDataTcp.fc),' Read ITF'));	

END_IF;
END_GET
END_PROPERTY

PROPERTY NoTcpAccesSince : TIME
GET
NoTcpAccesSince := tNoTcpAccesSince;
END_GET
END_PROPERTY

PROPERTY P_Tcp_fbstInterface : CtaSysConfig.ITF_STRING40
GET
P_Tcp_fbstInterface := scParameter.scTcp.fbstInterface;
END_GET
END_PROPERTY

PROPERTY P_Tcp_fbtWatchDog : CtaSysConfig.ITF_TIME
GET
P_Tcp_fbtWatchDog := scParameter.scTcp.fbtWatchDog;
END_GET
END_PROPERTY

PROPERTY P_LoggingOp : CtaSysConfig.ITF_DWORD
GET
P_LoggingOp := scParameter.loggingOp;
END_GET
END_PROPERTY

END_FUNCTION_BLOCK

// 30 Program Organization Units/SERVER/Tcp/ServerTCP_Extended
FUNCTION_BLOCK ServerTCP_Extended EXTENDS ModbusFB.ServerTCP
VAR_INPUT
END_VAR
VAR_OUTPUT
END_VAR
VAR
	_reqData : ModbusFB.RequestData;
END_VAR

SUPER^();

PROPERTY RequestData : ModbusFB.RequestData
GET
RequestData := _reqData;
END_GET
END_PROPERTY

(* Processes a MaskWriteRegister request.*)
METHOD PROTECTED ProcessMaskWriteRegister : ModbusFB.Error
VAR_IN_OUT CONSTANT
	(* The complete request data.*)
	reqData	: ModbusFB.RequestData;
END_VAR
VAR_IN_OUT
	(* Buffer to build the reply.*)
	replyBuffer	: ModbusFB.ByteBuffer;
END_VAR
VAR_OUTPUT
	(* Exception code eventually to reply.*)
	exceptionCode	: ModbusFB.ExceptionCodes;
END_VAR
ProcessMaskWriteRegister := SUPER^.ProcessMaskWriteRegister(reqData, replyBuffer, exceptionCode=>exceptionCode);
_reqData := reqData;
END_METHOD

//  Processes a ReadCoils request.
METHOD PROTECTED ProcessReadCoils : ModbusFB.Error
VAR_IN_OUT CONSTANT
	//  The complete request data.
	reqData : ModbusFB.RequestData;
END_VAR
VAR_IN_OUT
	//  Buffer to build the reply.
	replyBuffer : ModbusFB.ByteBuffer;
END_VAR
VAR_OUTPUT
	//  Exception code eventually to reply.
	exceptionCode : ModbusFB.ExceptionCodes;
END_VAR
ProcessReadCoils := SUPER^.ProcessReadCoils(reqData, replyBuffer, exceptionCode=>exceptionCode);
_reqData := reqData;
END_METHOD

(* Processes a ReadDiscreteInputs request.*)
METHOD PROTECTED ProcessReadDiscreteInputs : ModbusFB.Error
VAR_IN_OUT CONSTANT
	(* The complete request data.*)
	reqData	: ModbusFB.RequestData;
END_VAR
VAR_IN_OUT
	(* Buffer to build the reply.*)
	replyBuffer	: ModbusFB.ByteBuffer;
END_VAR
VAR_OUTPUT
	(* Exception code eventually to reply.*)
	exceptionCode	: ModbusFB.ExceptionCodes;
END_VAR
ProcessReadDiscreteInputs := SUPER^.ProcessReadDiscreteInputs(reqData, replyBuffer, exceptionCode=>exceptionCode);
_reqData := reqData;
END_METHOD

(* Processes a ReadHoldingRegisters request.*)
METHOD PROTECTED ProcessReadHoldingRegisters : ModbusFB.Error
VAR_IN_OUT CONSTANT
	(* The complete request data.*)
	reqData	: ModbusFB.RequestData;
END_VAR
VAR_IN_OUT
	(* Buffer to build the reply.*)
	replyBuffer	: ModbusFB.ByteBuffer;
END_VAR
VAR_OUTPUT
	(* Exception code eventually to reply.*)
	exceptionCode	: ModbusFB.ExceptionCodes;
END_VAR
ProcessReadHoldingRegisters := SUPER^.ProcessReadHoldingRegisters(reqData, replyBuffer, exceptionCode=>exceptionCode);
_reqData := reqData;
END_METHOD

(* Processes a ReadInputRegisters request.*)
METHOD PROTECTED ProcessReadInputRegisters : ModbusFB.Error
VAR_IN_OUT CONSTANT
	(* The complete request data.*)
	reqData	: ModbusFB.RequestData;
END_VAR
VAR_IN_OUT
	(* Buffer to build the reply.*)
	replyBuffer	: ModbusFB.ByteBuffer;
END_VAR
VAR_OUTPUT
	(* Exception code eventually to reply.*)
	exceptionCode	: ModbusFB.ExceptionCodes;
END_VAR
ProcessReadInputRegisters := SUPER^.ProcessReadInputRegisters(reqData, replyBuffer, exceptionCode=>exceptionCode);
_reqData := reqData;
END_METHOD

METHOD PROTECTED ProcessReadWriteMultipleRegisters : ModbusFB.Error
VAR_IN_OUT CONSTANT
	(* Request data already read from requestBuffer.*)
	reqData	: ModbusFB.RequestData;
END_VAR
VAR_IN_OUT
	(* Request buffer, reqData read already, write data remaining in request buffer.*)
	requestBuffer	: ModbusFB.ByteBuffer;
	(* Buffer to build the reply.*)
	replyBuffer	: ModbusFB.ByteBuffer;
END_VAR
VAR_OUTPUT
	(* Exception code eventually to reply.*)
	exceptionCode	: ModbusFB.ExceptionCodes;
END_VAR
ProcessReadWriteMultipleRegisters := SUPER^.ProcessReadWriteMultipleRegisters(reqData,requestBuffer, replyBuffer, exceptionCode=>exceptionCode);
_reqData := reqData;
END_METHOD

(* Processes a WriteMultipleCoils request.*)
METHOD PROTECTED ProcessWriteMultipleCoils : ModbusFB.Error
VAR_IN_OUT CONSTANT
	(* Request data already read from requestBuffer.*)
	reqData	: ModbusFB.RequestData;
END_VAR
VAR_IN_OUT
	(* Request buffer, reqData read already, write data remaining in request buffer.*)
	requestBuffer	: ModbusFB.ByteBuffer;
	(* Buffer to build the reply.*)
	replyBuffer	: ModbusFB.ByteBuffer;
END_VAR
VAR_OUTPUT
	(* Exception code eventually to reply.*)
	exceptionCode	: ModbusFB.ExceptionCodes;
END_VAR
ProcessWriteMultipleCoils := SUPER^.ProcessWriteMultipleCoils(reqData,requestBuffer, replyBuffer, exceptionCode=>exceptionCode);
_reqData := reqData;
END_METHOD

(* Processes a WriteMultipleRegisters request.*)
METHOD PROTECTED ProcessWriteMultipleRegisters : ModbusFB.Error
VAR_IN_OUT CONSTANT
	(* Request data already read from requestBuffer.*)
	reqData	: ModbusFB.RequestData;
END_VAR
VAR_IN_OUT
	(* Request buffer, reqData read already, write data remaining in request buffer.*)
	requestBuffer	: ModbusFB.ByteBuffer;
	(* Buffer to build the reply.*)
	replyBuffer	: ModbusFB.ByteBuffer;
END_VAR
VAR_OUTPUT
	(* Exception code eventually to reply.*)
	exceptionCode	: ModbusFB.ExceptionCodes;
END_VAR
ProcessWriteMultipleRegisters := SUPER^.ProcessWriteMultipleRegisters(reqData,requestBuffer, replyBuffer, exceptionCode=>exceptionCode);
_reqData := reqData;
END_METHOD

(* Processes a WriteSingleCoil request.*)
METHOD PROTECTED ProcessWriteSingleCoil : ModbusFB.Error
VAR_IN_OUT CONSTANT
	(* Request data already read from requestBuffer.*)
	reqData	: ModbusFB.RequestData;
END_VAR
VAR_IN_OUT
	(* Request buffer, reqData read already, write data remaining in request buffer.*)
	requestBuffer	: ModbusFB.ByteBuffer;
	(* Buffer to build the reply.*)
	replyBuffer	: ModbusFB.ByteBuffer;
END_VAR
VAR_OUTPUT
	(* Exception code eventually to reply.*)
	exceptionCode	: ModbusFB.ExceptionCodes;
END_VAR
ProcessWriteSingleCoil := SUPER^.ProcessWriteSingleCoil(reqData,requestBuffer, replyBuffer, exceptionCode=>exceptionCode);
_reqData := reqData;
END_METHOD

(* Processes a WriteSingleRegister request.*)
METHOD PROTECTED ProcessWriteSingleRegister : ModbusFB.Error
VAR_IN_OUT CONSTANT
	(* Request data already read from requestBuffer.*)
	reqData	: ModbusFB.RequestData;
END_VAR
VAR_IN_OUT
	(* Request buffer, reqData read already, write data remaining in request buffer.*)
	requestBuffer	: ModbusFB.ByteBuffer;
	(* Buffer to build the reply.*)
	replyBuffer	: ModbusFB.ByteBuffer;
END_VAR
VAR_OUTPUT
	(* Exception code eventually to reply.*)
	exceptionCode	: ModbusFB.ExceptionCodes;
END_VAR
ProcessWriteSingleRegister := SUPER^.ProcessWriteSingleRegister(reqData,requestBuffer, replyBuffer, exceptionCode=>exceptionCode);
_reqData := reqData;
END_METHOD

END_FUNCTION_BLOCK

// 30 Program Organization Units/SERVER/Serial/ServerSerial_Extended
FUNCTION_BLOCK ServerSerial_Extended EXTENDS ModbusFB.ServerSerial
VAR_INPUT
END_VAR
VAR_OUTPUT
END_VAR
VAR
	_reqData : ModbusFB.RequestData;
END_VAR

SUPER^(xEnable := xEnable AND NOT xError AND NOT xInactive );

PROPERTY RequestData : ModbusFB.RequestData
GET
RequestData := _reqData;
END_GET
END_PROPERTY

(* Processes a MaskWriteRegister request.*)
METHOD PROTECTED ProcessMaskWriteRegister : ModbusFB.Error
VAR_IN_OUT CONSTANT
	(* The complete request data.*)
	reqData	: ModbusFB.RequestData;
END_VAR
VAR_IN_OUT
	(* Buffer to build the reply.*)
	replyBuffer	: ModbusFB.ByteBuffer;
END_VAR
VAR_OUTPUT
	(* Exception code eventually to reply.*)
	exceptionCode	: ModbusFB.ExceptionCodes;
END_VAR
ProcessMaskWriteRegister := SUPER^.ProcessMaskWriteRegister(reqData, replyBuffer, exceptionCode=>exceptionCode);
_reqData := reqData;
END_METHOD

//  Processes a ReadCoils request.
METHOD PROTECTED ProcessReadCoils : ModbusFB.Error
VAR_IN_OUT CONSTANT
	//  The complete request data.
	reqData : ModbusFB.RequestData;
END_VAR
VAR_IN_OUT
	//  Buffer to build the reply.
	replyBuffer : ModbusFB.ByteBuffer;
END_VAR
VAR_OUTPUT
	//  Exception code eventually to reply.
	exceptionCode : ModbusFB.ExceptionCodes;
END_VAR
ProcessReadCoils := SUPER^.ProcessReadCoils(reqData, replyBuffer, exceptionCode=>exceptionCode);
_reqData := reqData;
END_METHOD

(* Processes a ReadDiscreteInputs request.*)
METHOD PROTECTED ProcessReadDiscreteInputs : ModbusFB.Error
VAR_IN_OUT CONSTANT
	(* The complete request data.*)
	reqData	: ModbusFB.RequestData;
END_VAR
VAR_IN_OUT
	(* Buffer to build the reply.*)
	replyBuffer	: ModbusFB.ByteBuffer;
END_VAR
VAR_OUTPUT
	(* Exception code eventually to reply.*)
	exceptionCode	: ModbusFB.ExceptionCodes;
END_VAR
ProcessReadDiscreteInputs := SUPER^.ProcessReadDiscreteInputs(reqData, replyBuffer, exceptionCode=>exceptionCode);
_reqData := reqData;
END_METHOD

(* Processes a ReadHoldingRegisters request.*)
METHOD PROTECTED ProcessReadHoldingRegisters : ModbusFB.Error
VAR_IN_OUT CONSTANT
	(* The complete request data.*)
	reqData	: ModbusFB.RequestData;
END_VAR
VAR_IN_OUT
	(* Buffer to build the reply.*)
	replyBuffer	: ModbusFB.ByteBuffer;
END_VAR
VAR_OUTPUT
	(* Exception code eventually to reply.*)
	exceptionCode	: ModbusFB.ExceptionCodes;
END_VAR
ProcessReadHoldingRegisters := SUPER^.ProcessReadHoldingRegisters(reqData, replyBuffer, exceptionCode=>exceptionCode);
_reqData := reqData;
END_METHOD

(* Processes a ReadInputRegisters request.*)
METHOD PROTECTED ProcessReadInputRegisters : ModbusFB.Error
VAR_IN_OUT CONSTANT
	(* The complete request data.*)
	reqData	: ModbusFB.RequestData;
END_VAR
VAR_IN_OUT
	(* Buffer to build the reply.*)
	replyBuffer	: ModbusFB.ByteBuffer;
END_VAR
VAR_OUTPUT
	(* Exception code eventually to reply.*)
	exceptionCode	: ModbusFB.ExceptionCodes;
END_VAR
ProcessReadInputRegisters := SUPER^.ProcessReadInputRegisters(reqData, replyBuffer, exceptionCode=>exceptionCode);
_reqData := reqData;
END_METHOD

METHOD PROTECTED ProcessReadWriteMultipleRegisters : ModbusFB.Error
VAR_IN_OUT CONSTANT
	(* Request data already read from requestBuffer.*)
	reqData	: ModbusFB.RequestData;
END_VAR
VAR_IN_OUT
	(* Request buffer, reqData read already, write data remaining in request buffer.*)
	requestBuffer	: ModbusFB.ByteBuffer;
	(* Buffer to build the reply.*)
	replyBuffer	: ModbusFB.ByteBuffer;
END_VAR
VAR_OUTPUT
	(* Exception code eventually to reply.*)
	exceptionCode	: ModbusFB.ExceptionCodes;
END_VAR
ProcessReadWriteMultipleRegisters := SUPER^.ProcessReadWriteMultipleRegisters(reqData,requestBuffer, replyBuffer, exceptionCode=>exceptionCode);
_reqData := reqData;
END_METHOD

(* Processes a WriteMultipleCoils request.*)
METHOD PROTECTED ProcessWriteMultipleCoils : ModbusFB.Error
VAR_IN_OUT CONSTANT
	(* Request data already read from requestBuffer.*)
	reqData	: ModbusFB.RequestData;
END_VAR
VAR_IN_OUT
	(* Request buffer, reqData read already, write data remaining in request buffer.*)
	requestBuffer	: ModbusFB.ByteBuffer;
	(* Buffer to build the reply.*)
	replyBuffer	: ModbusFB.ByteBuffer;
END_VAR
VAR_OUTPUT
	(* Exception code eventually to reply.*)
	exceptionCode	: ModbusFB.ExceptionCodes;
END_VAR
ProcessWriteMultipleCoils := SUPER^.ProcessWriteMultipleCoils(reqData,requestBuffer, replyBuffer, exceptionCode=>exceptionCode);
_reqData := reqData;
END_METHOD

(* Processes a WriteMultipleRegisters request.*)
METHOD PROTECTED ProcessWriteMultipleRegisters : ModbusFB.Error
VAR_IN_OUT CONSTANT
	(* Request data already read from requestBuffer.*)
	reqData	: ModbusFB.RequestData;
END_VAR
VAR_IN_OUT
	(* Request buffer, reqData read already, write data remaining in request buffer.*)
	requestBuffer	: ModbusFB.ByteBuffer;
	(* Buffer to build the reply.*)
	replyBuffer	: ModbusFB.ByteBuffer;
END_VAR
VAR_OUTPUT
	(* Exception code eventually to reply.*)
	exceptionCode	: ModbusFB.ExceptionCodes;
END_VAR
ProcessWriteMultipleRegisters := SUPER^.ProcessWriteMultipleRegisters(reqData,requestBuffer, replyBuffer, exceptionCode=>exceptionCode);
_reqData := reqData;
END_METHOD

(* Processes a WriteSingleCoil request.*)
METHOD PROTECTED ProcessWriteSingleCoil : ModbusFB.Error
VAR_IN_OUT CONSTANT
	(* Request data already read from requestBuffer.*)
	reqData	: ModbusFB.RequestData;
END_VAR
VAR_IN_OUT
	(* Request buffer, reqData read already, write data remaining in request buffer.*)
	requestBuffer	: ModbusFB.ByteBuffer;
	(* Buffer to build the reply.*)
	replyBuffer	: ModbusFB.ByteBuffer;
END_VAR
VAR_OUTPUT
	(* Exception code eventually to reply.*)
	exceptionCode	: ModbusFB.ExceptionCodes;
END_VAR
ProcessWriteSingleCoil := SUPER^.ProcessWriteSingleCoil(reqData,requestBuffer, replyBuffer, exceptionCode=>exceptionCode);
_reqData := reqData;
END_METHOD

(* Processes a WriteSingleRegister request.*)
METHOD PROTECTED ProcessWriteSingleRegister : ModbusFB.Error
VAR_IN_OUT CONSTANT
	(* Request data already read from requestBuffer.*)
	reqData	: ModbusFB.RequestData;
END_VAR
VAR_IN_OUT
	(* Request buffer, reqData read already, write data remaining in request buffer.*)
	requestBuffer	: ModbusFB.ByteBuffer;
	(* Buffer to build the reply.*)
	replyBuffer	: ModbusFB.ByteBuffer;
END_VAR
VAR_OUTPUT
	(* Exception code eventually to reply.*)
	exceptionCode	: ModbusFB.ExceptionCodes;
END_VAR
ProcessWriteSingleRegister := SUPER^.ProcessWriteSingleRegister(reqData,requestBuffer, replyBuffer, exceptionCode=>exceptionCode);
_reqData := reqData;
END_METHOD

END_FUNCTION_BLOCK

// 21 Interface/CLIENT/RTU/ITF_MB_CLIENT_RTU
INTERFACE ITF_MB_CLIENT_RTU  EXTENDS ITF_CLIENT

PROPERTY TIMEOUT : TIME
GET
END_GET
END_PROPERTY

PROPERTY WRITE_DELAY : TIME
GET
END_GET
END_PROPERTY

PROPERTY NODE_ID : USINT
GET
END_GET
END_PROPERTY

PROPERTY P_fbtReadDelay : CtaSysConfig.ITF_DATATYPE
GET
END_GET
END_PROPERTY

PROPERTY P_fbtWriteDelay : CtaSysConfig.ITF_DATATYPE
GET
END_GET
END_PROPERTY

PROPERTY P_fbusiNodeId : CtaSysConfig.ITF_DATATYPE
GET
END_GET
END_PROPERTY

PROPERTY P_fbxEnable : CtaSysConfig.ITF_DATATYPE
GET
END_GET
END_PROPERTY

PROPERTY P_fbtTimeOut : CtaSysConfig.ITF_DATATYPE
GET
END_GET
END_PROPERTY

PROPERTY READ_DELAY : TIME
GET
END_GET
END_PROPERTY

END_INTERFACE

// 30 Program Organization Units/FC/fcSetInitialIPString
FUNCTION fcSetInitialIPString : BOOL
VAR_INPUT
    ITF_STRING40In : CtaSysConfig.ITF_STRING40;	
END_VAR
VAR
END_VAR

IF __QUERYINTERFACE(ITF_STRING40In,ITF_STRING40In) THEN
    IF ITF_STRING40In.proValue = '' THEN    
        ITF_STRING40In.proValue := '0.0.0.0';
    END_IF;
    fcSetInitialIPString := TRUE;
ELSE
    fcSetInitialIPString := FALSE;
END_IF;

END_FUNCTION

// 30 Program Organization Units/SERVER/fbModBusServer
{warning 'Each Modbus server needs 400000 bytes of dynamic memory'}
FUNCTION_BLOCK fbModBusServer IMPLEMENTS ITF_SERVER
VAR_INPUT
    I_SerialPort                    :   WagoTypesCom.I_WagoSysComBase;
END_VAR
VAR_OUTPUT
    xError                          :   BOOL;
END_VAR
VAR
    (* Memory *)
    ayxCoil                         :   POINTER TO ARRAY[0..16#FFFF] OF BOOL;
    ayxDiscretInput                 :   POINTER TO ARRAY[0..16#FFFF] OF BOOL;  
    aywInputRegister                :   POINTER TO ARRAY[0..16#FFFF] OF WORD;
    aywHoldingRegister              :   POINTER TO ARRAY[0..16#FFFF] OF WORD; 
    xMemoryError                    :   BOOL;
    xMemoryAllocate                 :   BOOL    := TRUE;
    (* Tcp *)
    fbMbServerModelTcp              :   WagoAppPlcModbus.FbMbSlaveDataModel;
    fbMbShowAccesTcp                :   WagoAppPlcModbus.FbShowMbAccessInfo;
    fbMbTcpServer                   :   WagoAppPlcModbus.FbMbServerTcp;
    scKeepAlive                     :   WagoAppPlcModbus.typKeepAlive;
    ltLastAccesTcp                  :   LTIME;
    fbLastAccesTcp                  :   CtaAppTime.fbTimeMeasurement;
    xErrorWatchDogTcp               :   BOOL;
    xErrorTcp                       :   BOOL;
    
    (* Udp *)
    fbMbServerModelUdp              :   WagoAppPlcModbus.FbMbSlaveDataModel;
    fbMbShowAccesUdp                :   WagoAppPlcModbus.FbShowMbAccessInfo;
    fbMbUdpServer                   :   WagoAppPlcModbus.fbMbServerUdp;
    ltLastAccesUdp                  :   LTIME;
    fbLastAccesUdp                  :   CtaAppTime.fbTimeMeasurement;  
    xErrorWatchDogUdp               :   BOOL;  
    xErrorUdp                       :   BOOL;
    
    (* Serial *)
    fbMbServerModelSerial           :   WagoAppPlcModbus.FbMbSlaveDataModel;
    fbMbShowAccesSerial             :   WagoAppPlcModbus.FbShowMbAccessInfo;
    fbMbRtuSerialServer             :   WagoAppPlcModbus.FbMbServerSerial;
    ltLastAccesSerial               :   LTIME;
    fbLastAccesSerial               :   CtaAppTime.fbTimeMeasurement;
    xErrorWatchDogSerial            :   BOOL;    
    xErrorSerial                    :   BOOL;
    
    (* Parameter *)
    fbConfigFile                    :   CtaSysConfig.fbConfigFile;
    scParameter                     :   scModBusServerParameter;
END_VAR

actConfig();
IF xMemoryAllocate AND NOT xMemoryError THEN
    ayxCoil             := __NEW(BOOL,16#10000);
    ayxDiscretInput     := __NEW(BOOL,16#10000);
    aywInputRegister    := __NEW(WORD,16#10000);
    aywHoldingRegister  := __NEW(WORD,16#10000);
    IF ayxCoil <> 0 AND ayxDiscretInput <> 0 AND aywInputRegister <> 0 AND aywHoldingRegister <> 0 THEN
        xMemoryAllocate     := FALSE;     
    ELSE 
        xMemoryError := TRUE;   
    END_IF;
END_IF;
IF  NOT xMemoryAllocate AND NOT xMemoryError THEN
    IF SIZEOF(ayxCoil^) = 65536 AND SIZEOF(ayxDiscretInput^) = 65536 AND SIZEOF(aywInputRegister^) = 131072 AND SIZEOF(aywHoldingRegister^) = 131072 THEN
        IF NOT fbConfigFile.xError THEN
            actModBusServerSerial();
            actModBusServerTcp();
            actModBusServerUdp();
        END_IF;    
        xMemoryError := FALSE;
    ELSE
        xMemoryError := TRUE;    
    END_IF
END_IF;
(* Error *)
xError := fbConfigFile.xError OR xErrorTcp OR xErrorUdp OR xErrorSerial OR xMemoryError;

ACTION actConfig:
(* Config File *)
fbConfigFile();

scParameter.scSerial.fbbyUnitId            (_usiParaNr :=  1, ItfConfigFb := fbConfigFile , _MinInit :=    0     , _MaxInit :=     247 ); 
scParameter.scSerial.fbxEnable             (_usiParaNr :=  2, ItfConfigFb := fbConfigFile                                              );
scParameter.scSerial.fbudiBaudrate         (_usiParaNr :=  3, ItfConfigFb := fbConfigFile , _MinInit := 9600     , _MaxInit :=   19600 );
scParameter.scSerial.fbusiDataBits         (_usiParaNr :=  4, ItfConfigFb := fbConfigFile , _MinInit :=    5     , _MaxInit :=       8 );
scParameter.scSerial.fbiParity             (_usiParaNr :=  5, ItfConfigFb := fbConfigFile , _MinInit :=    0     , _MaxInit :=       5 );
scParameter.scSerial.fbiStopBits           (_usiParaNr :=  6, ItfConfigFb := fbConfigFile , _MinInit :=    0     , _MaxInit :=       5 );
scParameter.scSerial.fbiHandshake          (_usiParaNr :=  7, ItfConfigFb := fbConfigFile , _MinInit :=    0     , _MaxInit :=       7 );
scParameter.scSerial.fbiPhysikal           (_usiParaNr :=  8, ItfConfigFb := fbConfigFile , _MinInit :=    0     , _MaxInit :=       6 );
scParameter.scSerial.fbxRtuOrAscii         (_usiParaNr :=  9, ItfConfigFb := fbConfigFile                                              );
scParameter.scSerial.fbxEnableWatchDog     (_usiParaNr := 10, ItfConfigFb := fbConfigFile                                              );
scParameter.scSerial.fbtWatchDog           (_usiParaNr := 11, ItfConfigFb := fbConfigFile , _MinInit := T#1S     , _MaxInit :=   T#10M );
scParameter.scTcp.fbxEnable                (_usiParaNr := 12, ItfConfigFb := fbConfigFile                                              );
scParameter.scTcp.fbbyUnitId               (_usiParaNr := 13, ItfConfigFb := fbConfigFile , _MinInit :=    0     , _MaxInit :=     255 ); 
scParameter.scTcp.fbwPort                  (_usiParaNr := 14, ItfConfigFb := fbConfigFile , _MinInit :=    0     , _MaxInit := 16#FFFF );
scParameter.scTcp.fbxKeepAlive             (_usiParaNr := 15, ItfConfigFb := fbConfigFile                                              );
scParameter.scTcp.fbtMaxIdleTime           (_usiParaNr := 16, ItfConfigFb := fbConfigFile , _MinInit := T#1S     , _MaxInit :=   T#10M );
scParameter.scTcp.fbtIntervall             (_usiParaNr := 17, ItfConfigFb := fbConfigFile , _MinInit := T#1S     , _MaxInit :=   T#10M );
scParameter.scTcp.fbudiProbes              (_usiParaNr := 18, ItfConfigFb := fbConfigFile , _MinInit :=    0     , _MaxInit :=     500 );
scParameter.scTcp.fbxEnableWatchDog        (_usiParaNr := 19, ItfConfigFb := fbConfigFile                                              );
scParameter.scTcp.fbtWatchDog              (_usiParaNr := 20, ItfConfigFb := fbConfigFile , _MinInit := T#50MS   , _MaxInit :=   T#10M );
scParameter.scUdp.fbxEnable                (_usiParaNr := 21, ItfConfigFb := fbConfigFile                                              );
scParameter.scUdp.fbbyUnitId               (_usiParaNr := 22, ItfConfigFb := fbConfigFile , _MinInit :=    0     , _MaxInit :=     255 ); 
scParameter.scUdp.fbwPort                  (_usiParaNr := 23, ItfConfigFb := fbConfigFile , _MinInit :=    0     , _MaxInit := 16#FFFF );
scParameter.scUdp.fbxEnableWatchDog        (_usiParaNr := 24, ItfConfigFb := fbConfigFile                                              );
scParameter.scUdp.fbtWatchDog              (_usiParaNr := 25, ItfConfigFb := fbConfigFile , _MinInit := T#1S     , _MaxInit :=   T#10M );
END_ACTION

ACTION actModBusServerSerial:
(* Server Memory Serial*)
fbMbServerModelSerial(  bUnitId             := scParameter.scSerial.fbbyUnitId.byValue,
                        IIdentifyObject     := GVL_CtaModBus.fbDeviceName,
                        axDiscreteInputs    := ayxDiscretInput^,
                        axCoils             := ayxCoil^,
                        awInputRegisters    := aywInputRegister^,
                        awHoldingRegisters  := aywHoldingRegister^);  
                        
(* SERIAL Server *)           
IF scParameter.scSerial.fbxEnable.xValue THEN    
	IF __QUERYINTERFACE(I_SerialPort,I_SerialPort) THEN
		(* Server Run*) 
		fbMbRtuSerialServer(xConnect            := scParameter.scSerial.fbxEnable.xValue,
							I_Port              := I_SerialPort,
							udiBaudrate         := scParameter.scSerial.fbudiBaudrate.udiValue,
							usiDataBits         := scParameter.scSerial.fbusiDataBits.usiValue,
							eParity             := scParameter.scSerial.fbiParity.iValue,
							eStopBits           := scParameter.scSerial.fbiStopBits.iValue,
							eHandshake          := scParameter.scSerial.fbiHandshake.iValue,
							ePhysical           := scParameter.scSerial.fbiPhysikal.iValue,
							eFrameType          := SEL(scParameter.scSerial.fbxRtuOrAscii.xValue,WagoAppPlcModbus.eMbFrameType.RTU,WagoAppPlcModbus.eMbFrameType.ASCII),
							I_MbDataModel       := fbMbServerModelSerial.I_MbDataModel);
   	END_IF;                     
    (* Acces Info *)
    fbMbShowAccesSerial (   oMbAccessInfo := fbMbServerModelSerial.oMbAccessInfo); 
    
    (* Acces Time *)
    IF fbMbServerModelSerial.isReadAccess OR fbMbServerModelSerial.isWriteAccess THEN
        fbLastAccesSerial.Start();
        ltLastAccesSerial := fbLastAccesSerial.Stop();
    ELSE
        ltLastAccesSerial := fbLastAccesSerial.Stop();
    END_IF;
    
    (* WatchDog *)
    IF scParameter.scSerial.fbxEnableWatchDog.xValue THEN
        xErrorWatchDogSerial := TO_LTIME(scParameter.scSerial.fbtWatchDog.tValue) < ltLastAccesSerial;
    ELSE
        xErrorWatchDogSerial := FALSE;
    END_IF;                        
                        
ELSIF fbMbRtuSerialServer.xConnect THEN
    (* Server Disconnect *)
    fbMbRtuSerialServer(xConnect            := FALSE,
                        I_Port              := I_SerialPort,
                        I_MbDataModel       := fbMbServerModelSerial.I_MbDataModel);   
ELSE
    xErrorWatchDogSerial := FALSE;
    ltLastAccesSerial    := fbLastAccesSerial.Stop();
END_IF;                        



(* Error *)
xErrorSerial := fbConfigFile.xError OR fbMbServerModelSerial.xError OR fbMbRtuSerialServer.xError OR xErrorWatchDogSerial;
END_ACTION

ACTION actModBusServerTcp:
(* Server Memory Tcp*)
fbMbServerModelTcp(     bUnitId             := scParameter.scTcp.fbbyUnitId.byValue,
                        IIdentifyObject     := GVL_CtaModBus.fbDeviceName,
                        axDiscreteInputs    := ayxDiscretInput^,
                        axCoils             := ayxCoil^,
                        awInputRegisters    := aywInputRegister^,
                        awHoldingRegisters  := aywHoldingRegister^); 
                        
(* Tcp Server *)
IF scParameter.scTcp.fbxEnable.xValue THEN
    scKeepAlive.xEnable                     := scParameter.scTcp.fbxKeepAlive.xValue;
    scKeepAlive.tMaxIdleTime                := scParameter.scTcp.fbtMaxIdleTime.tValue;
    scKeepAlive.tInterval                   := scParameter.scTcp.fbtIntervall.tValue;
    scKeepAlive.udiProbes                   := scParameter.scTcp.fbudiProbes.udiValue;
    fbMbTcpServer(      xOpen               := scParameter.scTcp.fbxEnable.xValue,
                        wPort               := scParameter.scTcp.fbwPort.wValue,
                        utKeepAlive         := scKeepAlive,
                        eFrameType          := WagoAppPlcModbus.eMbFrameType.ETHERNET,
                        I_MbDataModel       := fbMbServerModelTcp.I_MbDataModel);
ELSIF fbMbTcpServer.xOpen THEN
    fbMbTcpServer(      xOpen               := FALSE,
                        I_MbDataModel       := fbMbServerModelTcp.I_MbDataModel);                           
END_IF;                        

(* Acces Info *)
fbMbShowAccesTcp    (   oMbAccessInfo := fbMbServerModelTcp.oMbAccessInfo);   

(* Acces Time *)
IF fbMbServerModelTcp.isReadAccess OR fbMbServerModelTcp.isWriteAccess THEN
    fbLastAccesTcp.Start();
    ltLastAccesTcp := fbLastAccesTcp.Stop();
ELSE
    ltLastAccesTcp := fbLastAccesTcp.Stop();
END_IF;

(* WatchDog *)
IF scParameter.scTcp.fbxEnableWatchDog.xValue THEN
    xErrorWatchDogTcp := TO_LTIME(scParameter.scTcp.fbtWatchDog.tValue) < ltLastAccesTcp;
ELSE
    xErrorWatchDogTcp := FALSE;
END_IF;

(* Error *)
xErrorTcp := fbConfigFile.xError OR fbMbServerModelTcp.xError OR fbMbTcpServer.xError OR xErrorWatchDogTcp;
END_ACTION

ACTION actModBusServerUdp:
(* Server Memory Udp*)
fbMbServerModelUdp(     bUnitId             := scParameter.scUdp.fbbyUnitId.byValue,
                        IIdentifyObject     := GVL_CtaModBus.fbDeviceName,
                        axDiscreteInputs    := ayxDiscretInput^,
                        axCoils             := ayxCoil^,
                        awInputRegisters    := aywInputRegister^,
                        awHoldingRegisters  := aywHoldingRegister^);  
                        
(* UDP Server *)
IF scParameter.scUdp.fbxEnable.xValue THEN
    fbMbUdpServer(      xOpen               := scParameter.scUdp.fbxEnable.xValue,
                        wPort               := scParameter.scUdp.fbwPort.wValue,
                        eFrameType          := WagoAppPlcModbus.eMbFrameType.ETHERNET,
                        I_MbDataModel       := fbMbServerModelUdp.I_MbDataModel);
ELSIF fbMbUdpServer.xOpen THEN
    fbMbUdpServer(      xOpen               := FALSE,
                        I_MbDataModel       := fbMbServerModelUdp.I_MbDataModel);                        
END_IF;                          

(* Acces Info *)
fbMbShowAccesUdp    (   oMbAccessInfo := fbMbServerModelUdp.oMbAccessInfo); 

(* Acces Time *)
IF fbMbServerModelUdp.isReadAccess OR fbMbServerModelUdp.isWriteAccess THEN
    fbLastAccesUdp.Start();
    ltLastAccesUdp := fbLastAccesSerial.Stop();
ELSE
    ltLastAccesUdp := fbLastAccesSerial.Stop();
END_IF;

(* WatchDog *)
IF scParameter.scUdp.fbxEnableWatchDog.xValue THEN
    xErrorWatchDogUdp := TO_LTIME(scParameter.scUdp.fbtWatchDog.tValue) < ltLastAccesUdp;
ELSE
    xErrorWatchDogUdp := FALSE;
END_IF;

(* Error *)
xErrorUdp := fbConfigFile.xError OR fbMbServerModelUdp.xError OR fbMbUdpServer.xError OR xErrorWatchDogUdp;
END_ACTION

METHOD metAddSerialControll : BOOL
VAR_INPUT
    I_DataAccesListener :   WagoAppPlcModbus.I_DataAccessListener;
END_VAR
fbMbServerModelSerial.RegisterDataAccessListener(I_DataAccesListener);
END_METHOD

METHOD metAddTcpControll : BOOL
VAR_INPUT
    I_DataAccesListener :   WagoAppPlcModbus.I_DataAccessListener;
END_VAR
fbMbServerModelTcp.RegisterDataAccessListener(I_DataAccesListener);
END_METHOD

METHOD metAddUdpControll : BOOL
VAR_INPUT
    I_DataAccesListener :   WagoAppPlcModbus.I_DataAccessListener;
END_VAR
fbMbServerModelUdp.RegisterDataAccessListener(I_DataAccesListener);
END_METHOD

METHOD metGetCoil : BOOL
VAR_INPUT
    wAdr          : WORD;
END_VAR
IF NOT xMemoryAllocate AND NOT xMemoryError THEN
	IF wAdr >= LOWER_BOUND(ayxCoil^,1) AND wAdr <= UPPER_BOUND(ayxCoil^,1) THEN
    	metGetCoil := ayxCoil^[wAdr];
	END_IF;
END_IF;
END_METHOD

METHOD metGetHoldingRegister : WORD
VAR_INPUT
    wAdr          : WORD;
END_VAR
IF NOT xMemoryAllocate AND NOT xMemoryError THEN
	IF wAdr >= LOWER_BOUND(aywHoldingRegister^,1) AND wAdr <= UPPER_BOUND(aywHoldingRegister^,1) THEN
    	metGetHoldingRegister := aywHoldingRegister^[wAdr];
	END_IF;
END_IF;
END_METHOD

METHOD metSetCoil : BOOL
VAR_INPUT
    wAdr          : WORD;
    xValue        : BOOL;
END_VAR
IF NOT xMemoryAllocate AND NOT xMemoryError THEN
	IF wAdr >= LOWER_BOUND(ayxCoil^,1) AND wAdr <= UPPER_BOUND(ayxCoil^,1) THEN
    	ayxCoil^[wAdr] := xValue;
	END_IF;
END_IF;
END_METHOD

METHOD metSetDiscretInput : BOOL
VAR_INPUT
    wAdr          : WORD;
    xValue        : BOOL;
END_VAR
IF NOT xMemoryAllocate AND NOT xMemoryError THEN
	IF wAdr >= LOWER_BOUND(ayxDiscretInput^,1) AND wAdr <= UPPER_BOUND(ayxDiscretInput^,1) THEN
    	ayxDiscretInput^[wAdr] := xValue;
	END_IF;
END_IF;
END_METHOD

METHOD metSetHoldingRegister : BOOL
VAR_INPUT
    wAdr          : WORD;
    wValue        : WORD;
END_VAR
IF NOT xMemoryAllocate AND NOT xMemoryError THEN
	IF wAdr >= LOWER_BOUND(aywHoldingRegister^,1) AND wAdr <= UPPER_BOUND(aywHoldingRegister^,1) THEN
    	aywHoldingRegister^[wAdr] := wValue;
	END_IF;
END_IF;
END_METHOD

METHOD metSetInputRegister : BOOL
VAR_INPUT
    wAdr          : WORD;
    wValue        : WORD;
END_VAR
IF NOT xMemoryAllocate AND NOT xMemoryError THEN
	IF wAdr >= LOWER_BOUND(aywInputRegister^,1) AND wAdr <= UPPER_BOUND(aywInputRegister^,1) THEN
    	aywInputRegister^[wAdr] := wValue;
	END_IF;
END_IF;
END_METHOD

END_FUNCTION_BLOCK

// 30 Program Organization Units/CLIENT/BASE/FB_MB_CLIENT
FUNCTION_BLOCK FB_MB_CLIENT EXTENDS CtaAppBmk.fbBMK IMPLEMENTS ITF_CLIENT
VAR_OUTPUT
	udiDynMem					:	UDINT;
	xAllJobsDone				:	BOOL;
	xConfirmAllJobsDone			:	BOOL;
END_VAR             			
VAR                 			
	_ITF_BIG_SYBIL				:	ITF_CLIENT;
	_ITF_LOW_SYBIL				:	ITF_CLIENT;
	                			
	_BASE_MBU_JOB				:	ITF_MBJOB;
	_TEMP_REG_JOB				:	ITF_MBJOB;
	_TEMP_MBU_JOB				:	ITF_MBJOB;	
	
	_COUNT						:	UINT;
	_udiDynMemTemp				:	UDINT;
	xGetReadyCalled				:	BOOL;
	xNoChangeHappen				:	BOOL;
	xDestroyAllJobs				:	BOOL;
	
	xErrorHappen				:	BOOL;
	eErrorID					:	ModbusFB.Error;
	eExeptionCode				:	ModbusFB.ExceptionCodes;
	
	fbTimeStop					:	CtaAppTime.fbTimeMeasurement;
	ltTime						:	LTIME;
	
	_ayITF_MBJOB_VIS			:	ARRAY[0..9] OF ITF_MBJOB;
END_VAR

PROPERTY ENABLE : BOOL
GET
ENABLE := FALSE;
END_GET
END_PROPERTY

